(* CODESYS project p6lib-common.library
   Company: MacGregor
   DefaultNamespace: p6com
   Version: 1.1.4
   DocFormat: reStructuredText
   Placeholder: p6lib_common
   Title: p6lib_common

Project tree, tasks and I/O mapping:
  libraries: p7lib-basetypes, * (MacGregor); Tc2_EtherCAT, * (Beckhoff Automation GmbH); Tc2_Math, * (Beckhoff Automation GmbH); Tc2_Standard, * (Beckhoff Automation GmbH); Tc2_System, * (Beckhoff Automation GmbH); Tc2_Utilities, * (Beckhoff Automation GmbH); Tc3_EventLogger, * (Beckhoff Automation GmbH); Tc3_Module, * (Beckhoff Automation GmbH)
  AnalogOut/
    DUT/
      data type EL40xxIO_out
    function block AnalogOutBiPolarScalableAA [ST]: processing
    function block AnalogOutEL40xx [ST]: processing, Value
    function block AnalogOutPercentAA [ST]: processing
    function block AnalogOutUniPolarScalableAA [ST]: processing
    OutputClassCatalog.txt
  00000000-0000-0000-0000-000000000000|AnalogOut\OutputClassCatalog.txt
  ByteAndBits/
    function ClearBit16 [ST]
    function ClearBit8 [ST]
    function Get_LSB_From_UINT [ST]
    function Get_LSB_From_Word [ST]
    function Get_MSB_From_UINT [ST]
    function Get_MSB_From_Word [ST]
    function GetBit16 [ST]
    function GetBit8 [ST]
    function SetBit16 [ST]
    function SetBit8 [ST]
  Concurrency/
    interface IMutex: acquire, acquired, context, isAcquiredByMe, release
    function block Mutex [ST]: acquire, acquired, context, isAcquiredByMe, release
  counter/
    function block CounterExpansion [ST]: FromDINT_TO_LINT
  Cycle Time/
    function block CycleTime [ST]: Cycletime, update
  EmergencyStop/
    DUT/
      data type ConfigEmergencyStop
      data type EStopSM
    function block EmergencyStop [ST]: Activated, ActivatedSwitchIdx, ActivatedSwitchName, ExternEStop, GroupError, resetGroupError
  EventManagement/
    DUT/
      data type AlarmTable
      data type EventProcessing
    function block AlarmAnalog [ST]: _createArguments, _processing, _processPipeline
    function block AlarmAnalogValueHigh [ST]: _processPipeline
    function block AlarmAnalogValueLow [ST]: _processPipeline
    function block AlarmCollector [ST]: AlarmCritical, AlarmWarning, ConfirmAlarms, OnAlarmConfirmed, OnAlarmRaised, reset, update
    function block AlarmCollectorEx [ST]: AlarmCritical, AlarmWarning, ConfirmAlarms, copyTableToHMI, delEvent, Execute, getText, insertEvent, OnAlarmCleared, OnAlarmConfirmed, OnAlarmRaised, reset
    function block AlarmDigital [ST]
    function block AlarmDigitalEx [ST]: _createArguments
    function block AlarmEvent [ST]: _createArguments, _createEvent, clear, confirm, FB_init, raise, Raised
    function block AlarmOilFilter [ST]
    function block AlarmSensorError [ST]
    function block AlarmSensorValueHigh [ST]: _processPipeline
    function block AlarmSensorValueLow [ST]: _processPipeline
    function block AlarmSimple [ST]
    function block StartupDelay [ST]: Done, FB_init
  Fieldbus/
    DUT/
      data type CU2508StatIO_In
      data type EFieldbusQueryResult
      data type ESimpleFieldbusSM
      data type EthercatCoEObject
      data type EthercatCoEObjectArray
      data type EthercatCoEValueArray
      data type EthTypes
      data type EthValue
      data type EthWriteCoEArraySM
    function block Ethercat [ST]: _readCoEData, _writeCoEData, isDevice, readCoEDataBYTE, readCoEDataDINT, readCoEDataDWORD, readCoEDataINT, readCoEDataLINT, readCoEDataLREAL, readCoEDataLWORD, readCoEDataREAL, readCoEDataSINT, readCoEDataUDINT, readCoEDataUINT, readCoEDataULINT, readCoEDataUSINT, readCoEDataWORD, readCoEValueArray, wait, writeCoEDataBYTE, writeCoEDataDINT, writeCoEDataDWORD, writeCoEDataINT, writeCoEDataLINT, writeCoEDataLREAL, writeCoEDataLWORD, writeCoEDataREAL, writeCoEDataSINT, writeCoEDataUDINT, writeCoEDataUINT, writeCoEDataULINT, writeCoEDataUSINT, writeCoEDataWORD, writeCoEValueArray
    function block EthercatCU2508Stat [ST]: getLostFrames, setNull
    function block EthercatMasterStat [ST]: LostFrames, setNull
  IOHandler/
    interface IIOHandler: get
    function block IOHandler [ST]: FB_init, get
  Math/
    function CosineRuleKnownAllSides [ST]
    function CosineRuleKnownAnAngle [ST]
    function HorizontalLength [ST]
    function Scale [ST]
    function Signum [ST]
    function VerticalHeight [ST]
  MRU/
    DUT/
      data type ConfigMRU
    interface IMRUReader: DataAvailable, getData
    function block MRU [ST]: getValues, transform, update
  NMEA/
    DUT/
      data type TNMEAint
      data type TNMEAreal
      data type TNMEAsentence
      data type TNMEAstring
      data type TNMEAStructDescription
    function block NMEA_TrawlLength [ST]
    function block NMEA_TrawlSpeed [ST]
    function block NMEA_TrawlTension [ST]
    function block NMEAParser [ST]: _hexChkSum_to_byte, _incp, calcChkSum, getChkSumFromSentence, getHeader, getIntField, getRealField, getStringField, parse, setFieldsOfInterest
    function block NMEASentence [ST]: calcCheckSum, DataOut, formatSentenceWith3Values
    function block NMEATransmitter6021 [ST]: Busy
  ObjectProtocols/
    DUT/
    V1/
      function block ProtoBase1ToN [ST]: attach, FB_init, getNoServices, getService, getServiceByIdx, isAttached, resetService, setService
      function block ProtoBaseNTo1 [ST]: attach, FB_init, getMaster, getMasterByIdx, getNoMasters, isAttached, resetServices, setMaster
      function block ProtoMasterSingleService [ST]: attach, getService
  OperationTime/
    DUT/
      data type OperationTimeSM
    function block DeviceOpTime [ST]: Optime
    function block OperationTimeCounter [ST]: reset, update
  ParameterManagment/
    AddParameter/
      function block AddParameterBool [ST]
      function block AddParameterInt [ST]
      function block AddParameterLreal [ST]
      function block AddParameterStr [ST]
      function block AddParameterTime [ST]
    DUT/
      data type DataType
      data type ParameterList
  PID/
    DUT/
    function block HTrawlController [ST]: ErrorPosition, ErrorVelocity, Tension, TorqueOut
    function block HTrawlController2 [ST]: CtrlLimit, ErrorPosition, ErrorVelocity, Tension, TorqueOut, VelocitySetpoint
    function block HTrawlController3 [ST]: CtrlLimit, ErrorPosition, ErrorVelocity, Tension, TorqueOut, VelocitySetpoint
    function block HTrawlController4 [ST]: CtrlLimit, ErrorPosition, ErrorVelocity, Tension, TorqueOut, VelocitySetpoint
    function block HTrawlController5 [ST]: CtrlLimit, ErrorPosition, ErrorVelocity, Tension, TorqueOut, VelocitySetpoint
    function block HTrawlController6 [ST]: CtrlLimit, ErrorPosition, ErrorVelocity, Tension, TorqueOut, VelocitySetpoint
    function block PIDController [ST]: Error, Out, update
    function block PIDController2P [ST]: Error, Out, update
    function block PIDControllerLINT [ST]: Error, Out, update
  Sensor/
    DUT/
      data type BarthUnsignedIO_In
      data type EL30xxIO_in
      data type EL30xxStatus
      data type EL30xxStatusWordBit
      data type SensorBinaryIO_in
    Fishpump/
      DUT/
        data type SensorBarthIO_In
      function block SensorBarthBase [ST]: Error, processing, Value, ValueRaw
      function block SensorBarthPressure [ST]: processing
      function block SensorBarthTemp [ST]: processing
      function block SensorBarthUnsigned [ST]: processing
    HandlingBody/
      function block AnglePosition [ST]: processing
      function block StrokePosition [ST]: Angle, Height, Length, processing, Stroke
      data type StrokePositionConfig
    HydPressure/
      data type AnglePositionConfig
      function block HydPressure250barAA [ST]: processing
      function block HydPressure60barAA [ST]: processing
    OilFilter/
      function block OilFilterSensor [ST]: Error, processing, Value, ValueRaw
    Pressure/
      function block Pressure10barAA [ST]: processing
    Scalable/
      function block Sensor20mAA [ST]: processing
      function block SensorASymRangeAA [ST]: processing
      function block SensorSymRange [ST]: processing
      function block SensorSymRangeAA [ST]: processing
    Temperature/
      function block TempSensorAB [ST]: processing
      function block TempSensorAC [ST]: processing
      function block TempSensorAA [ST]: processing
    function block DummySensor [ST]: Error, Value, ValueRaw
    SensorCatalog.txt
    function block SensorEL30xx [ST]: Error, processing, Value, ValueRaw
  00000000-0000-0000-0000-000000000000|Sensor\SensorCatalog.txt
  SignalClassifier/
    DUT/
    function block SignalClassGTEQ [ST]: processing, Signal, update
    function block SignalClassLTEQ [ST]: processing, Signal, update
  SignalProcessing/
    DUT/
      data type SwitchHysteresisSM
    function block Filter1stDeg [ST]
    function block Filter1stDegEx [ST]: reset
    function block InverseOneSideTest [ST]
    interface ISignalPipeline: analogAbs, analogFilter1stDeg, analogLimitBand, analogLimitLowerBoundary, analogLimitUpperBoundary, analogReversePolarity, analogScale, boolInverse, boolTestTimeSpan, getAnalogValue, getBinaryValue, retrieveValues, setBoolInput, setLRealInput, testFalling, testGreaterOrEqual, testLessOrEqual, testRaising
    function block OneSideTest [ST]
    function block SignalPipeline [ST]: analogAbs, analogFilter1stDeg, analogLimitBand, analogLimitLowerBoundary, analogLimitUpperBoundary, analogReversePolarity, analogScale, boolInverse, boolTestTimeSpan, getAnalogValue, getBinaryValue, retrieveValues, setBoolInput, setLRealInput, testFalling, testGreaterOrEqual, testLessOrEqual, testRaising
    function block TwoSideTest [ST]
  Signals/
    function block OneShotSignal [ST]: Get, Set
    function block OneShotSignalInt [ST]: Get, Set
  TimingGenerators/
    function block CycleGenerator [ST]: Q, update
    function block CycleTimer [ST]
    function block SymmetricPulse [ST]: Value
  UnitConversion/
    DUT/
      data type ConfigSystemUnits
      data type LengthUnits
      data type TensionUnits
      data type VelocityUnits
    function block UnitConverter [ST]: getLengthUnit, getTensionUnit, getVelocityUnit, kgToUnit, meterToUnit, MSToUnit, unitToKg, unitToMeter, unitToMS
  global variables Parameters
*)

// AnalogOut/DUT/EL40xxIO_out
TYPE EL40xxIO_out :
	STRUCT
		output	: INT;
	END_STRUCT
END_TYPE

// EmergencyStop/DUT/ConfigEmergencyStop
TYPE ConfigEmergencyStop :
	STRUCT
		switchname : ARRAY[0..Parameters.SizeOfEStopArray-1] OF P6IdName;
	END_STRUCT
END_TYPE

// EmergencyStop/DUT/EStopSM
{attribute 'qualified_only'}
{attribute 'strict'}
TYPE EStopSM :
	(
		STARTUP 			:= 0,
		WAITRESET			:= 10,
		IDLE				:= 20,
		ESTOP				:= 30,
		ESTOP_RELEASED		:= 40,
		GRP_RST_START		:= 50,
		GRP_RST_EXE			:= 60, 
		GRP_RST_END			:= 70
	) INT;
END_TYPE

// EventManagement/DUT/AlarmTable
TYPE AlarmTable :
	STRUCT
		eventID : UDINT;
		timestamp : STRING;
		message : STRING(255);
	END_STRUCT
END_TYPE

// EventManagement/DUT/EventProcessing
TYPE EventProcessing :
	STRUCT
		event : REFERENCE TO FB_TcEvent;
		uid : UDINT;
		eventID : UDINT;
		timestamp : STRING;
		message : STRING(255);
		hasTxt : BOOL;
	END_STRUCT
END_TYPE

// Fieldbus/DUT/CU2508StatIO_In
TYPE CU2508StatIO_In :
	STRUCT
		addr : ARRAY[0..7] OF AMSNETID;
	END_STRUCT
END_TYPE

// Fieldbus/DUT/EFieldbusQueryResult
{attribute 'qualified_only'}
{attribute 'strict'}
TYPE EFieldbusQueryResult :
(
	OK 					:= 0,
	FAIL				:= -1,
	BUSY				:= 1
) INT;
END_TYPE

// Fieldbus/DUT/ESimpleFieldbusSM
{attribute 'qualified_only'}
{attribute 'strict'}
TYPE ESimpleFieldbusSM :
(
	IDLE			:= 0,
	STARTUP			:= 1,
	WAITONRESULT	:= 2,
	RESULT			:= 3			
) INT;
END_TYPE

// Fieldbus/DUT/EthercatCoEObject
TYPE EthercatCoEObject :
	STRUCT
		para	: DWORD := 16#FFFF_FFFF; // Format XXXXYY X: Parameter group, Y: Parameter. Has no functionality other than to provide data for the HMI and to mark the end of the list
		idx		: WORD;
		sidx	: BYTE;  
		tclass 	: EthTypes := EthTypes.TWORD;	
	END_STRUCT
END_TYPE

// Fieldbus/DUT/EthercatCoEObjectArray
TYPE 
	EthercatCoEObjectArray : ARRAY[0..Parameters.SizeOfEthCoEValues-1] OF EthercatCoEObject; 
END_TYPE

// Fieldbus/DUT/EthercatCoEValueArray
TYPE 
	EthercatCoEValueArray : ARRAY[0..Parameters.SizeOfEthCoEValues-1] OF EthValue; 
END_TYPE

// Fieldbus/DUT/EthTypes
{attribute 'qualified_only'}
{attribute 'strict'}
TYPE EthTypes :
(
	TWORD			:= 0,
	TBYTE			:= 1,
	TDWORD			:= 2,
	TLWORD			:= 3,
	TSINT			:= 4,
	TUSINT			:= 5,
	TINT			:= 6,
	TUINT			:= 7,
	TDINT			:= 8,
	TUDINT			:= 9,
	TLINT			:= 10,
	TULINT			:= 11,
	TREAL			:= 12,
	TLREAL			:= 13
) INT;
END_TYPE

// Fieldbus/DUT/EthValue
TYPE EthValue :
	UNION
		VBYTE			: BYTE;
		VWORD			: WORD;
		VDWORD			: DWORD;
		VLWORD			: LWORD;
		VSINT			: SINT;
		VUSINT			: USINT;
		VINT			: INT;
		VUINT			: UINT;
		VDINT			: DINT;
		VUDINT			: UDINT;
		VLINT			: LINT;
		VULINT			: ULINT;
		VREAL			: REAL;
		VLREAL			: LREAL;
	END_UNION
END_TYPE

// Fieldbus/DUT/EthWriteCoEArraySM
{attribute 'qualified_only'}
{attribute 'strict'}
TYPE EthWriteCoEArraySM :
(
	IDLE		 	:= 0,
	WRITE			:= 10,
	ERROR			:= 20,
	READY			:= 30,
	INCR			:= 40
) INT;
END_TYPE

// MRU/DUT/ConfigMRU
TYPE ConfigMRU :
	STRUCT
		Option_Transformation		: BOOL := FALSE;
		Option_Reverse_Position 	: BOOL := FALSE;
		Option_Reverse_Velocity 	: BOOL := FALSE;
		Option_Reverse_Acceleration : BOOL := FALSE;
		Option_Reverse_Roll			: BOOL := FALSE;
		Option_Reverse_Ritch		: BOOL := FALSE;
		Option_MRUSet				: INT  := -1; // Values for coordinate set from 0..9, when transformation is used
				
		// Section Transformation 					
		CycleTime 					: LREAL := 0.05; // Cycletime of the MRU in sec
		FilterAcceleration			: LREAL := 1.0; // Values from 0..1!
		PosX						: ARRAY[0..19] OF LREAL; // X axis forward aligned
		PosY 						: ARRAY[0..19] OF LREAL; // Y axis port aliged
		PosZ						: ARRAY[0..19] OF LREAL; // Z upwards aligned
	END_STRUCT
END_TYPE

// NMEA/DUT/TNMEAint
TYPE TNMEAint : LINT; END_TYPE

// NMEA/DUT/TNMEAreal
TYPE TNMEAreal : LREAL; END_TYPE

// NMEA/DUT/TNMEAsentence
TYPE TNMEAsentence : STRING(254); END_TYPE

// NMEA/DUT/TNMEAstring
TYPE TNMEAstring : STRING(128); END_TYPE

// NMEA/DUT/TNMEAStructDescription
TYPE TNMEAStructDescription : STRING(32); END_TYPE

// OperationTime/DUT/OperationTimeSM
{attribute 'qualified_only'}
{attribute 'strict'}
TYPE OperationTimeSM :
(
	IDLE 		:= 0,
	ACTIVE		:= 1
);
END_TYPE

// ParameterManagment/DUT/DataType
TYPE DataType :
	STRUCT
		intType : INT;
		boolType : BOOL;
		stringType : STRING;
		lrealType : LREAL;
		timeType : TIME;
	END_STRUCT
END_TYPE

// ParameterManagment/DUT/ParameterList
TYPE ParameterList :
	STRUCT
		name : STRING := 'Ω FREE';
		value : DataType;
		unit : STRING;
		status : STRING;
	END_STRUCT
END_TYPE

// Sensor/DUT/BarthUnsignedIO_In
TYPE BarthUnsignedIO_In :
	STRUCT
		input	: INT;
	END_STRUCT
END_TYPE

// Sensor/DUT/EL30xxIO_in
TYPE EL30xxIO_in :
	STRUCT
		status 	: EL30xxStatus;
		input	: INT;
	END_STRUCT
END_TYPE

// Sensor/DUT/EL30xxStatus
TYPE EL30xxStatus :
	UNION
		twobyte : WORD;
		bits 	: EL30xxStatusWordBit;
	END_UNION
END_TYPE

// Sensor/DUT/EL30xxStatusWordBit
TYPE EL30xxStatusWordBit :
	STRUCT
		UnderRange			: BIT;		// 0
		OverRange			: BIT;		// 1
		Limit1				: BIT;		// 2
		Limit2				: BIT;		// 3
		Reserved4			: BIT;		// 4
		Reserved5			: BIT;		// 5
		Error				: BIT;		// 6
		Reserved7			: BIT;		// 7
		Reserved8			: BIT;		// 8
		Reserved9			: BIT;		// 9	
		Reserved10			: BIT;		// 10
		Reserved11			: BIT;		// 11
		Reserved12			: BIT;		// 12
		Reserved13			: BIT;		// 13
		Reserved14			: BIT;		// 14
		Reserved15			: BIT;		// 15
	END_STRUCT
END_TYPE

// Sensor/DUT/SensorBinaryIO_in
TYPE SensorBinaryIO_in :
	STRUCT
		signal	: BOOL; 
	END_STRUCT
END_TYPE

// Sensor/Fishpump/DUT/SensorBarthIO_In
TYPE SensorBarthIO_In :
	STRUCT
		input	: WORD;
	END_STRUCT
END_TYPE

// Sensor/HandlingBody/StrokePositionConfig
TYPE StrokePositionConfig :
	STRUCT
		FilterCoefficient : LREAL := 0.1;// 1stDegFilter, cant be 0.
		CalibratedLowerLimit : LREAL;	//min sensor measurement
		CalibratedUpperLimit : LREAL;	//max sensor measurement
		MinStroke : LREAL;
		MaxStroke : LREAL;
		CylinderToNextJointMin : LREAL;
		CylinderToNextJointMax : LREAL;	
		
		BoltToBoltLength : LREAL;
		BoltToCylinderBoltLength : LREAL;
		TiltLegLength : LREAL;
		InverseDirection : BOOL;
	END_STRUCT
END_TYPE

// Sensor/HydPressure/AnglePositionConfig
TYPE AnglePositionConfig :
	STRUCT
		FilterCoefficient : LREAL := 0.1;// 1stDegFilter, cant be 0.
		CalibratedLowerLimit : LREAL;	//min sensor measurement
		CalibratedUpperLimit : LREAL;	//max sensor measurement
		MaxAngle : LREAL;		// [deg]total range this joint operate in
	END_STRUCT
END_TYPE

// SignalProcessing/DUT/SwitchHysteresisSM
{attribute 'qualified_only'}
{attribute 'strict'}
TYPE SwitchHysteresisSM :
(
	START 			:= 0,
	IDLE			:= 10,
	ON				:= 20,
	WAITFOROFF		:= 30,
	BANDUP			:= 40,
	BANDDOWN		:= 50 
) INT;
END_TYPE

// UnitConversion/DUT/ConfigSystemUnits
TYPE ConfigSystemUnits :
	STRUCT
		velocityUnit : VelocityUnits;
		tensionUnit  : TensionUnits;
		lengthUnit   : LengthUnits;
	END_STRUCT
END_TYPE

// UnitConversion/DUT/LengthUnits
{attribute 'qualified_only'}
{attribute 'strict'}
TYPE LengthUnits :
(
	METER 	:= 0,
	FEET 	:= 1,
	FATHOM 	:= 2
) DINT;
END_TYPE

// UnitConversion/DUT/TensionUnits
{attribute 'qualified_only'}
{attribute 'strict'}
TYPE TensionUnits :
(
	KILO 		:= 0,
	TON_METRIC	:= 1,
	TON_IMPERIAL:= 2,
	POUND 		:= 3
) DINT;
END_TYPE

// UnitConversion/DUT/VelocityUnits
{attribute 'qualified_only'}
{attribute 'strict'}
TYPE VelocityUnits :
(
	METER_PER_SEC 	:= 0,
	METER_PER_MIN 	:= 1,
	FEET_PER_MIN 	:= 2,
	FATHOM_PER_MIN	:= 3
) DINT;
END_TYPE

// Parameters
{attribute 'qualified_only'}
VAR_GLOBAL CONSTANT
	SizeOfEthCoEValues 	: INT := 200;
	SizeOfEStopArray	: INT := 100;
	
	//
	// This is related to protocol definitions
	//
	ServicesPerMaster	: DINT := 100;
	MastersPerService	: DINT := 100;
END_VAR

// AnalogOut/AnalogOutBiPolarScalableAA
(* 
	Use this class only, when the scaling values are unknown!
*)
FUNCTION_BLOCK AnalogOutBiPolarScalableAA EXTENDS AnalogOutEL40xx IMPLEMENTS IAnalogOut
VAR_INPUT
	ValueMax	: LREAL;
	ValueMin	: LREAL;
END_VAR
VAR
	{attribute 'hide'} 
	pipe			: SignalPipeline;
END_VAR

SUPER^();
THIS^.processing();

METHOD PROTECTED  processing : BOOL
VAR_INST
	val : LREAL;
END_VAR
IF ABS(ValueMax-ValueMin)>=0.1 THEN
	val :=  THIS^.pipe
						.setLRealInput(THIS^.rvalue)
						.analogScale(ValueMin, ValueMax, THIS^.ADC_VALUE_MIN, THIS^.ADC_VALUE_MAX, TRUE)
						.getAnalogValue();
								
	THIS^.IO_Out.output := LREAL_TO_INT(val);
ELSE
	THIS^.IO_Out.output := 0;	
END_IF
END_METHOD

END_FUNCTION_BLOCK

// AnalogOut/AnalogOutEL40xx
FUNCTION_BLOCK ABSTRACT AnalogOutEL40xx
VAR_INPUT
	IO_Out					: REFERENCE TO EL40xxIO_Out;
END_VAR
VAR
	{attribute 'hide'} 
	rvalue					: LREAL;							
END_VAR
VAR CONSTANT
	{attribute 'hide'} 
	ADC_VALUE_MAX 			: LREAL := 16#7FFF;
	{attribute 'hide'} 
	ADC_VALUE_MIN 			: LREAL := 0;
END_VAR

METHOD PROTECTED ABSTRACT processing : BOOL
END_METHOD

{attribute 'monitoring' := 'call'}
{attribute 'TcRpcEnable'}
PROPERTY Value : LREAL
SET
rvalue := Value;
END_SET
END_PROPERTY

END_FUNCTION_BLOCK

// SignalProcessing/SignalPipeline
{attribute 'hide_all_locals'}
FUNCTION_BLOCK SignalPipeline IMPLEMENTS ISignalPipeline
VAR
	// Internal processing
	process_value_lreal				: LREAL;
	process_value_bool				: BOOL;
END_VAR

METHOD analogAbs : ISignalPipeline
VAR_INPUT
	Value 		: LREAL;
END_VAR
THIS^.process_value_lreal := ABS(THIS^.process_value_lreal);

analogAbs := THIS^;
END_METHOD

METHOD analogFilter1stDeg : ISignalPipeline
VAR_INPUT
	Coefficient				: LREAL;
END_VAR
VAR_INST
	_filter1stDeg 					: Filter1stDeg;	
END_VAR
_filter1stDeg( 
			Value:= THIS^.process_value_lreal, 
			Coefficient:= Coefficient, 
			Out => THIS^.process_value_lreal
		);

analogFilter1stDeg := THIS^;
END_METHOD

METHOD analogLimitBand : ISignalPipeline
VAR_INPUT
	BoundaryLower 		: LREAL;
	BoundaryUpper 		: LREAL;
END_VAR
THIS^.process_value_lreal := LIMIT(BoundaryLower, THIS^.process_value_lreal, BoundaryUpper);

analogLimitBand := THIS^;
END_METHOD

METHOD analogLimitLowerBoundary : ISignalPipeline
VAR_INPUT
	Boundary 		: LREAL;
END_VAR
THIS^.process_value_lreal := MAX(Boundary, THIS^.process_value_lreal);

analogLimitLowerBoundary := THIS^;
END_METHOD

METHOD analogLimitUpperBoundary : ISignalPipeline
VAR_INPUT
	Boundary 		: LREAL;
END_VAR
THIS^.process_value_lreal := MIN(Boundary, THIS^.process_value_lreal);

analogLimitUpperBoundary := THIS^;
END_METHOD

METHOD analogReversePolarity : ISignalPipeline
VAR_INPUT
	Enable : BOOL;
END_VAR
THIS^.process_value_lreal := SEL(Enable, THIS^.process_value_lreal, -THIS^.process_value_lreal);

analogReversePolarity := THIS^;
END_METHOD

METHOD analogScale : ISignalPipeline
VAR_INPUT
	InputMin 		: LREAL;
	InputMax		: LREAL;
	OutputMin		: LREAL;
	OutputMax		: LREAL;
	LimitOutput		: BOOL;
END_VAR
THIS^.process_value_lreal := Scale(
									Value 		:= THIS^.process_value_lreal,
									InputMin 	:= InputMin,
									InputMax	:= InputMax,
									OutputMin	:= OutputMin,
									OutputMax	:= OutputMax,
									LimitOutput	:= LimitOutput 
								);
								
analogScale := THIS^;
END_METHOD

METHOD boolInverse : ISignalPipeline

THIS^.process_value_bool := NOT THIS^.process_value_bool;

boolInverse := THIS^;
END_METHOD

METHOD boolTestTimeSpan : ISignalPipeline
VAR_INPUT
	TimeSpan	: TIME;
END_VAR
VAR_INST
	timerOn 	: TON;
END_VAR

timerOn(IN := THIS^.process_value_bool, PT := TimeSpan);

THIS^.process_value_bool := timerOn.Q;

boolTestTimeSpan := THIS^;
END_METHOD

METHOD getAnalogValue : LREAL

getAnalogValue := THIS^.process_value_lreal;
END_METHOD

METHOD getBinaryValue : BOOL

getBinaryValue := THIS^.process_value_bool;
END_METHOD

METHOD retrieveValues : ISignalPipeline
VAR_INPUT
	ValueLReal 	: REFERENCE TO LREAL;
	ValueBool	: REFERENCE TO BOOL;
END_VAR
IF  __ISVALIDREF(ValueLReal) THEN
	ValueLReal := THIS^.process_value_lreal;
END_IF

IF  __ISVALIDREF(ValueBool) THEN
	ValueBool := THIS^.process_value_bool;
END_IF

retrieveValues := THIS^;
END_METHOD

METHOD setBoolInput : ISignalPipeline
VAR_INPUT
	Value : BOOL;
END_VAR
THIS^.process_value_bool := Value;

setBoolInput := THIS^;
END_METHOD

(*
This method has to get the raw value and put into internal_processing_value 
when THIS^.retrieve = TRUE 
*)
METHOD setLRealInput : ISignalPipeline
VAR_INPUT
	Value	: LREAL;
END_VAR
THIS^.process_value_lreal := Value;
THIS^.process_value_bool := FALSE;


setLRealInput := THIS^;
END_METHOD

METHOD testFalling : ISignalPipeline
VAR_INST
	trigger : F_TRIG;
END_VAR
trigger(CLK := THIS^.process_value_bool, Q=>THIS^.process_value_bool);

testFalling := THIS^;
END_METHOD

METHOD testGreaterOrEqual : ISignalPipeline
VAR_INPUT
	Value		: LREAL;
	Hysteresis	: LREAL;
	MakeAnd		: BOOL;
END_VAR
VAR_INST
	oneside		: OneSideTest;
	res 		: BOOL;
END_VAR
oneside(
			Level := Value,
			Hysteresis := Hysteresis, 
			Value		:= THIS^.process_value_lreal,
			Out => res
		);
					
THIS^.process_value_bool := SEL(
								MakeAnd, 
								res OR THIS^.process_value_bool, 
								res AND THIS^.process_value_bool
							);
							
testGreaterOrEqual := THIS^;
END_METHOD

METHOD testLessOrEqual : ISignalPipeline
VAR_INPUT
	Value		: LREAL;
	Hysteresis	: LREAL;
	MakeAnd		: BOOL;
END_VAR
VAR_INST
	inv_oneside		: InverseOneSideTest;
	res 			: BOOL;
END_VAR
inv_oneside(
				Level 		:= Value,
				Hysteresis 	:= Hysteresis, 
				Value		:= THIS^.process_value_lreal,
				Out 		=> res
			);
					
THIS^.process_value_bool := SEL(
								MakeAnd, 
								res OR THIS^.process_value_bool, 
								res AND THIS^.process_value_bool
							);
							
							
testLessOrEqual := THIS^;
END_METHOD

METHOD testRaising : ISignalPipeline
VAR_INST
	trigger : R_TRIG;
END_VAR
trigger(CLK := THIS^.process_value_bool, Q=>THIS^.process_value_bool);

testRaising := THIS^;
END_METHOD

END_FUNCTION_BLOCK

// SignalProcessing/ISignalPipeline
INTERFACE ISignalPipeline

METHOD analogAbs : ISignalPipeline
VAR_INPUT
	Value 		: LREAL;
END_VAR
END_METHOD

METHOD analogFilter1stDeg : ISignalPipeline
VAR_INPUT
	Coefficient				: LREAL;
END_VAR
END_METHOD

METHOD analogLimitBand : ISignalPipeline
VAR_INPUT
	BoundaryLower 		: LREAL;
	BoundaryUpper 		: LREAL;
END_VAR
END_METHOD

METHOD analogLimitLowerBoundary : ISignalPipeline
VAR_INPUT
	Boundary 		: LREAL;
END_VAR
END_METHOD

METHOD analogLimitUpperBoundary : ISignalPipeline
VAR_INPUT
	Boundary 		: LREAL;
END_VAR
END_METHOD

METHOD analogReversePolarity : ISignalPipeline
VAR_INPUT
	Enable : BOOL;
END_VAR
END_METHOD

METHOD analogScale : ISignalPipeline
VAR_INPUT
	InputMin 		: LREAL;
	InputMax		: LREAL;
	OutputMin		: LREAL;
	OutputMax		: LREAL;
	LimitOutput		: BOOL;
END_VAR
END_METHOD

METHOD boolInverse : ISignalPipeline
END_METHOD

METHOD boolTestTimeSpan : ISignalPipeline
VAR_INPUT
	TimeSpan	: TIME;
END_VAR
END_METHOD

METHOD getAnalogValue : LREAL
END_METHOD

METHOD getBinaryValue : BOOL
END_METHOD

METHOD retrieveValues : ISignalPipeline
VAR_INPUT
	ValueLReal 	: REFERENCE TO LREAL;
	ValueBool	: REFERENCE TO BOOL;
END_VAR
END_METHOD

METHOD setBoolInput : ISignalPipeline
VAR_INPUT
	Value : BOOL;
END_VAR
END_METHOD

(*
This method has to get the raw value and put into internal_processing_value 
when THIS^.retrieve = TRUE 
*)
METHOD setLRealInput : ISignalPipeline
VAR_INPUT
	Value : LREAL;
END_VAR
END_METHOD

METHOD testFalling : ISignalPipeline
END_METHOD

METHOD testGreaterOrEqual : ISignalPipeline
VAR_INPUT
	Value		: LREAL;
	Hysteresis	: LREAL;
	MakeAnd		: BOOL;
END_VAR
END_METHOD

METHOD testLessOrEqual : ISignalPipeline
VAR_INPUT
	Value		: LREAL;
	Hysteresis	: LREAL;
	MakeAnd		: BOOL;
END_VAR
END_METHOD

METHOD testRaising : ISignalPipeline
END_METHOD

END_INTERFACE

// SignalProcessing/Filter1stDeg
(*
Purpose
=======
This is a 1st deg filter class. The coeffcient has a range from 0..1 and is limited automagically by this class

Methods And Properties
======================
*)
{attribute 'hide_all_locals'}
FUNCTION_BLOCK Filter1stDeg
VAR_INPUT
	Value 			: LREAL;
	Coefficient  	: LREAL;
END_VAR
VAR_OUTPUT
	Out 			: LREAL; 
END_VAR
VAR
	value_1 		: LREAL;
	value_0			: LREAL;
	CoefficientCopy : LREAL;
END_VAR


CoefficientCopy := LIMIT(0.0, Coefficient, 1.0);
value_0 := Value * CoefficientCopy + (1.0 - CoefficientCopy) * value_1; 

value_1 := value_0;

Out 	:= value_0;

END_FUNCTION_BLOCK

// Math/Scale
(*
This function is transposing an input range to an output range. The option of 
limiting output is for cases when a full range calibration isn't possible 
*)
{attribute 'hide_all_locals'}
FUNCTION Scale : LREAL
VAR_INPUT
	Value			: LREAL;
	InputMin 		: LREAL;
	InputMax 		: LREAL;
	OutputMin 		: LREAL;
	OutputMax 		: LREAL;
	LimitOutput : BOOL;
END_VAR
VAR
END_VAR

IF ((InputMax - InputMin) <> 0) THEN
	Scale := (OutputMax - OutputMin) / (InputMax - InputMin) * (Value - InputMin) + OutputMin;
	IF LimitOutput THEN
		IF OutputMax >= OutputMin THEN 
			Scale := LIMIT(OutputMin, Scale, OutputMax);
		ELSE
			Scale := LIMIT(OutputMax, Scale, OutputMin);			
		END_IF
	END_IF
ELSE
	Scale := 0;
END_IF

END_FUNCTION

// SignalProcessing/OneSideTest
(*
Purpose
=======
This class is a test whether a value is outside a range from 0 ..max. The max value has
a hysteresis



Methods And Properties
======================
*)
{attribute 'hide_all_locals'}
FUNCTION_BLOCK OneSideTest
VAR_INPUT
	Level	 	: LREAL;
	Hysteresis	: LREAL;
	Value		: LREAL;
END_VAR
VAR_OUTPUT
	Out			: BOOL;
END_VAR
VAR
	state : SwitchHysteresisSM;
END_VAR


CASE state OF 
	SwitchHysteresisSM.START:
		state := SwitchHysteresisSM.IDLE; 
		
	SwitchHysteresisSM.IDLE:
		IF Value >= Level + ABS(Hysteresis/2.0) THEN
			state := SwitchHysteresisSM.ON;
		END_IF
	
	SwitchHysteresisSM.ON:
		IF Value <= Level - ABS(Hysteresis/2.0) THEN
			state := SwitchHysteresisSM.IDLE;
		END_IF
	ELSE
		state := SwitchHysteresisSM.START;
END_CASE


Out := state = SwitchHysteresisSM.ON;

END_FUNCTION_BLOCK

// SignalProcessing/InverseOneSideTest
(*
Purpose
=======
This class is a test whether a value is outside a range from 0 ..max. The max value has
a hysteresis

Methods And Properties
======================
*)
{attribute 'hide_all_locals'}
FUNCTION_BLOCK InverseOneSideTest
VAR_INPUT
	Level	 	: LREAL;
	Hysteresis	: LREAL;
	Value		: LREAL;
END_VAR
VAR_OUTPUT
	Out 		: BOOL;
END_VAR
VAR
	state : SwitchHysteresisSM;
END_VAR


CASE state OF 
	SwitchHysteresisSM.START:
		state := SwitchHysteresisSM.IDLE; 
		
	SwitchHysteresisSM.IDLE:
		IF Value <= Level - ABS(Hysteresis/2.0) THEN
			state := SwitchHysteresisSM.ON;
		END_IF
	
	SwitchHysteresisSM.ON:
		IF Value >= Level + ABS(Hysteresis/2.0) THEN
			state := SwitchHysteresisSM.IDLE;
		END_IF
	ELSE
		state := SwitchHysteresisSM.START;
END_CASE


Out :=  state = SwitchHysteresisSM.ON;

END_FUNCTION_BLOCK

// AnalogOut/AnalogOutPercentAA
(* 
	Use this class only, when the scaling values are unknown!
*)
FUNCTION_BLOCK AnalogOutPercentAA EXTENDS AnalogOutEL40xx IMPLEMENTS IAnalogOut
VAR
	{attribute 'hide'} 
	pipe			: SignalPipeline;
END_VAR

SUPER^();
THIS^.processing();

METHOD PROTECTED  processing : BOOL
VAR_INST
	val : LREAL;
END_VAR
val :=  THIS^.pipe
							.setLRealInput(THIS^.rvalue)
							.analogScale(-1.0, 1.0, THIS^.ADC_VALUE_MIN, THIS^.ADC_VALUE_MAX, TRUE)
							.getAnalogValue();
							
THIS^.IO_Out.output := LREAL_TO_INT(val);
END_METHOD

END_FUNCTION_BLOCK

// AnalogOut/AnalogOutUniPolarScalableAA
(* 
	Use this class only, when the scaling values are unknown!
*)
FUNCTION_BLOCK AnalogOutUniPolarScalableAA EXTENDS AnalogOutEL40xx IMPLEMENTS IAnalogOut
VAR_INPUT
	ValueMax	: LREAL;
	ValueMin	: LREAL;
END_VAR
VAR
	{attribute 'hide'} 
	pipe			: SignalPipeline;
END_VAR

SUPER^();
THIS^.processing();

METHOD PROTECTED  processing : BOOL
VAR_INST
	val : LREAL;
END_VAR
IF ABS(ValueMax-ValueMin)>=0.1 THEN
	val :=  THIS^.pipe
								.setLRealInput(THIS^.rvalue)
								.analogScale(ValueMin, ValueMax, 0, THIS^.ADC_VALUE_MAX, TRUE)
								.getAnalogValue();
								
	THIS^.IO_Out.output := LREAL_TO_INT(val);
ELSE
	THIS^.IO_Out.output := 0;	
END_IF
END_METHOD

END_FUNCTION_BLOCK

// ByteAndBits/ClearBit16
FUNCTION ClearBit16 : WORD
VAR_INPUT
	Value 	: WORD;
	N  		: SINT;
END_VAR

ClearBit16 := DWORD_TO_WORD(ClearBit32(Value, N));

END_FUNCTION

// ByteAndBits/ClearBit8
FUNCTION ClearBit8 : BYTE
VAR_INPUT
	Value 	: BYTE;
	N  		: SINT;
END_VAR

ClearBit8 := DWORD_TO_BYTE(ClearBit32(Value, N));

END_FUNCTION

// ByteAndBits/Get_LSB_From_UINT
FUNCTION Get_LSB_From_UINT : USINT
VAR_INPUT
	data : UINT;
END_VAR
VAR
	{attribute 'hide'} 
	p : POINTER TO USINT;
END_VAR

p := ADR(data);
Get_LSB_From_UINT := p^;

END_FUNCTION

// ByteAndBits/Get_LSB_From_Word
FUNCTION Get_LSB_From_Word : BYTE
VAR_INPUT
	data : WORD;
END_VAR
VAR
	{attribute 'hide'} 
	p : POINTER TO BYTE;
END_VAR

p := ADR(data) ;
Get_LSB_From_Word := p^;

END_FUNCTION

// ByteAndBits/Get_MSB_From_UINT
FUNCTION Get_MSB_From_UINT : USINT;
VAR_INPUT
	data : UINT;
END_VAR
VAR
	{attribute 'hide'} 
	p : POINTER TO USINT;
END_VAR

p := ADR(data) + 1;
Get_MSB_From_UINT := p^;

END_FUNCTION

// ByteAndBits/Get_MSB_From_Word
FUNCTION Get_MSB_From_Word : BYTE
VAR_INPUT
	data : WORD;
END_VAR
VAR
	{attribute 'hide'} 
	p : POINTER TO BYTE;
END_VAR

p := ADR(data) + 1;
Get_MSB_From_Word := p^;

END_FUNCTION

// ByteAndBits/GetBit16
FUNCTION GetBit16 : BOOL
VAR_INPUT
	Value 	: WORD;
	N  		: SINT;
END_VAR

GetBit16 := GetBit32(Value, N);

END_FUNCTION

// ByteAndBits/GetBit8
FUNCTION GetBit8 : BOOL
VAR_INPUT
	Value 	: BYTE;
	N  		: SINT;	
END_VAR

GetBit8 := GetBit32(Value, N);

END_FUNCTION

// ByteAndBits/SetBit16
FUNCTION SetBit16 : WORD
VAR_INPUT
	Value 	: WORD;
	N  		: SINT;
END_VAR

SetBit16 := DWORD_TO_WORD(SetBit32(Value, N));

END_FUNCTION

// ByteAndBits/SetBit8
FUNCTION SetBit8 : BYTE;
VAR_INPUT
	Value 	: BYTE;
	N  		: SINT;
END_VAR

SetBit8 := DWORD_TO_BYTE(SetBit32(Value, N));

END_FUNCTION

// Concurrency/IMutex
INTERFACE IMutex

METHOD acquire : BOOL
VAR_INPUT
	Context : DINT;
END_VAR
END_METHOD

PROPERTY acquired : BOOL
GET
END_GET
END_PROPERTY

PROPERTY context : DINT
GET
END_GET
END_PROPERTY

METHOD isAcquiredByMe : BOOL
VAR_INPUT
	Context : DINT;
END_VAR
END_METHOD

METHOD release : BOOL
VAR_INPUT
	Context 	: DINT;
END_VAR
END_METHOD

END_INTERFACE

// Concurrency/Mutex
(*
Purpose
=======
This class is providing a Mutex functionality and is including a context identifier 

Methods And Properties
======================
*)
{attribute 'no_explicit_call' := 'do not call this POU directly'} 
FUNCTION_BLOCK Mutex
VAR
	{attribute 'hide'} 
	_acquired 		: BOOL;
	{attribute 'hide'} 
	_context		: DINT;
END_VAR

METHOD acquire : BOOL
VAR_INPUT
	Context : DINT;
END_VAR
IF NOT _acquired THEN
	acquire 	:= TRUE; 
	_acquired 	:= TRUE;
	_context	:= Context;
ELSE
	acquire 	:= FALSE; 
END_IF
END_METHOD

{attribute 'monitoring' := 'variable'}
PROPERTY acquired : BOOL
GET
acquired := _acquired;
END_GET
END_PROPERTY

{attribute 'monitoring' := 'variable'}
PROPERTY context : DINT
GET
context := _context;
END_GET
END_PROPERTY

METHOD isAcquiredByMe : BOOL
VAR_INPUT
	Context : DINT;
END_VAR

IF _acquired AND (Context = _context) THEN
	isAcquiredByMe := TRUE;
ELSE
	isAcquiredByMe := FALSE;	
END_IF
END_METHOD

METHOD release : BOOL
VAR_INPUT
	Context 	: DINT;
END_VAR
IF _acquired AND (Context=_context) THEN
	_acquired := FALSE;
	release := TRUE;
ELSE
	release := TRUE;	
END_IF
END_METHOD

END_FUNCTION_BLOCK

// counter/CounterExpansion
(*
	This class offers Counter Overflow prevention methods
*) 
FUNCTION_BLOCK CounterExpansion

METHOD FromDINT_TO_LINT : LINT
VAR_INPUT
	Counter 			: DINT;
	Overflow			: REFERENCE TO LINT;
END_VAR
VAR 
	past_counter		: LINT;
	actual_counter		: LINT;
	state 				: DINT;
END_VAR

past_counter := actual_counter;
actual_counter := counter;

CASE state OF 
	0: // no change in range
		IF (past_counter > 0)  AND  (actual_counter < 0) THEN 
			state := 1;
		ELSIF (past_counter < 0) AND (actual_counter > 0) THEN
			state := 2;
		END_IF
		
	1: // overflow on the top
		state := 0;
		Overflow := Overflow + LINT#16#1_0000_0000; 
		
	2: // overflow on the bottom
		state := 0;
		Overflow := Overflow - LINT#16#1_0000_0000; 
END_CASE

FromDINT_TO_LINT := actual_counter + Overflow;
END_METHOD

END_FUNCTION_BLOCK

// Cycle Time/CycleTime
(*
Purpose
=======
This class calculates the cycle time independent of a PLC supplier

Methods And Properties
======================
*)
{attribute 'no_explicit_call' := 'do not call this POU directly'} 
{attribute 'hide_all_locals'}
FUNCTION_BLOCK CycleTime
VAR
	t1, t0 : TIME;
	interval : UDINT;
	_cycletime : LREAL;	
END_VAR

{attribute 'monitoring' := 'variable'}
PROPERTY Cycletime : LREAL
GET
Cycletime := _Cycletime;
END_GET
END_PROPERTY

METHOD update : LREAL
t1 := t0; 

t0 := TIME();

interval := MIN(TIME_TO_UDINT(t0-t1), 100);

_cycletime := MAX(
					UDINT_TO_LREAL(interval)/1000.0,
					0.001
				);


update := _cycletime;
END_METHOD

END_FUNCTION_BLOCK

// EmergencyStop/EmergencyStop
FUNCTION_BLOCK EmergencyStop IMPLEMENTS p7type.IEmergencyStop;
VAR_INPUT
	Enabled									: BOOL;
	Config 									: REFERENCE TO ConfigEmergencyStop; 
END_VAR
VAR
	{attribute 'hide'} started 								: BOOL;
	{attribute 'hide'} state									: EStopSM;
	{attribute 'hide'} startUpTimer							: TON;
						grpResetStart						: TON;
						grpResetExe							: TON;
						grpResetEnd							: TON;
						cycleGen							: SymmetricPulse;
	
	{attribute 'hide'} _resetGroup								: BOOL;	
	{attribute 'hide'} _idx 									: INT;
	
	{attribute 'hide'} _switchIdx 								: INT;  //Switch identifier
	{attribute 'hide'} _switchName								: p7type.P6IdName;

	_EStopSwitches 			AT %I* 			: ARRAY [0..Parameters.SizeOfEStopArray-1] OF BOOL; //Emergency stop input
	_NoEStopDetected 		AT %I* 			: BOOL;	 //Emergency stop signal
	
	_ExternEStop 							: BOOL;
	_TwinSafe_Run 			AT %Q* 			: BOOL := TRUE;  //Run TwinSAFE logic
	_TwinSafeFB_Reset 		AT %Q*			: BOOL;	//Reset emergency stop
	_TwinSafeGroup_Reset	AT %Q*			: BOOL; //Group Reset	
	_TwinSafeGroupErrCom	AT %I*			: BOOL; // Group Com error
	_TwinSafeGroupErrFB		AT %I*			: BOOL; // Group FB Error
	_TwinSafeGroupErrOther	AT %I*			: BOOL; // Group Other Error	
END_VAR

IF NOT started THEN
	started := TRUE;
END_IF

cycleGen(CLK:=T#200MS);
_TwinSafeFB_Reset := cycleGen.Value;

startUpTimer(IN:=(state=EStopSM.WAITRESET), PT:=T#500MS);
grpResetStart(IN:=(state=EStopSM.GRP_RST_START), PT:=T#200MS);
grpResetExe(IN:=(state=EStopSM.GRP_RST_EXE), PT:=T#200MS);
grpResetEnd(IN:=(state=EStopSM.GRP_RST_END), PT:=T#200MS);


CASE state OF
	EStopSM.STARTUP:
		_TwinSafeGroup_Reset := TRUE;
		_TwinSafe_Run := TRUE;
		_resetGroup := FALSE;
		_switchName := '';
		_switchIdx := -1; //Emergency stop ok
		state := EStopSM.WAITRESET;
		
	EStopSM.WAITRESET:
		_TwinSafe_Run := TRUE;
		_TwinSafeGroup_Reset := FALSE;
		IF (NOT startUpTimer.Q) THEN
			state := EStopSM.GRP_RST_START;
		END_IF
	
	EStopSM.IDLE:
		_TwinSafe_Run := TRUE;
		_TwinSafeGroup_Reset := FALSE;
		IF (NOT _NoEStopDetected) AND Enabled THEN
			state := EStopSM.ESTOP;
		ELSIF _resetGroup THEN
			_resetGroup := FALSE;
			state := EStopSM.GRP_RST_START;
		END_IF
	
	EStopSM.ESTOP:
		_TwinSafe_Run := TRUE;
		_TwinSafeGroup_Reset := FALSE;
		IF _resetGroup THEN
			_resetGroup := FALSE;
			state := EStopSM.GRP_RST_START;
		ELSIF NOT _NoEStopDetected THEN
			_switchIdx := -1;
			// Find the first activated EStop switch 
			FOR _idx := 0 TO Parameters.SizeOfEStopArray-1 DO
				IF NOT _EStopSwitches[_idx] THEN
					_switchIdx := _idx;
					_switchName := Config.switchname[_idx];
					EXIT;
				END_IF
			END_FOR
		ELSE
			state := EStopSM.ESTOP_RELEASED;	
		END_IF
	
	EStopSM.ESTOP_RELEASED:
		_TwinSafe_Run := TRUE;
		_TwinSafeGroup_Reset := FALSE;
		_switchName := '';
		_switchIdx := -1;
		state := EStopSM.IDLE;
	
	ESTOPSM.GRP_RST_START:
		_TwinSafe_Run := FALSE;
		_TwinSafeGroup_Reset := FALSE;
		IF grpResetStart.Q THEN
			state := ESTOPSM.GRP_RST_EXE;
		END_IF
		
	ESTOPSM.GRP_RST_EXE:
		_TwinSafe_Run := FALSE;
		_TwinSafeGroup_Reset := TRUE;
		IF grpResetExe.Q THEN
			state := ESTOPSM.GRP_RST_END;
		END_IF

	ESTOPSM.GRP_RST_END:
		_TwinSafe_Run := FALSE;
		_TwinSafeGroup_Reset := FALSE;
		IF grpResetEnd.Q THEN
			state := ESTOPSM.IDLE;
		END_IF
END_CASE

{attribute 'monitoring' := 'call'}
{attribute 'TcRpcEnable'}
PROPERTY Activated : BOOL
GET
Activated := ((NOT _NoEStopDetected) OR _externEStop) AND Enabled;
END_GET
END_PROPERTY

{attribute 'monitoring' := 'call'}
{attribute 'TcRpcEnable'}
PROPERTY ActivatedSwitchIdx : INT
GET
ActivatedSwitchIdx := _switchIdx;
END_GET
END_PROPERTY

{attribute 'monitoring' := 'call'}
{attribute 'TcRpcEnable'}
PROPERTY ActivatedSwitchName : p7type.P6IdName
GET
ActivatedSwitchName := _switchName;
END_GET
END_PROPERTY

PROPERTY ExternEStop : BOOL
SET
_ExternEStop := ExternEStop;
END_SET
END_PROPERTY

{attribute 'monitoring' := 'call'}
{attribute 'TcRpcEnable'}
PROPERTY GroupError : BOOL
GET
GroupError := _TwinSafeGroupErrCom OR _TwinSafeGroupErrFB OR _TwinSafeGroupErrOther;
END_GET
END_PROPERTY

{attribute 'TcRpcEnable'}
METHOD resetGroupError : BOOL
_resetGroup := TRUE;
END_METHOD

END_FUNCTION_BLOCK

// TimingGenerators/SymmetricPulse
//Generates a pulse with 50% duty cycle
FUNCTION_BLOCK SymmetricPulse
VAR_INPUT
	CLK : TIME; // Time Period of signal. Signal is on CLK/2, and off CLK/2.
END_VAR
VAR_OUTPUT
END_VAR
VAR
	timer : TON;
	_value : BOOL;
END_VAR

timer(IN:=NOT timer.Q, PT:=CLK/2);
IF _value AND timer.Q THEN
	_value := FALSE;
ELSIF NOT _value AND timer.Q THEN
	_value := TRUE;
END_IF

PROPERTY Value : BOOL
GET
Value := _value;
END_GET
END_PROPERTY

END_FUNCTION_BLOCK

// EventManagement/AlarmAnalog
{attribute 'hide_all_locals'} 
FUNCTION_BLOCK ABSTRACT AlarmAnalog  EXTENDS AlarmEvent
VAR_INPUT
	LimitOn		: LREAL;
	LimitOff	: LREAL;
END_VAR
VAR
	_value		: LREAL;
	pipe		: SignalPipeline;
	distLimits	: LREAL;
END_VAR

_processing();

METHOD PROTECTED _createArguments : BOOL
SUPER^._createArguments();

THIS^.alarmEvt.ipArguments.AddLReal(_value);
END_METHOD

METHOD PROTECTED _processing : BOOL
VAR_INST
	state	: DINT;
	timerOn	: TON;
	timerOff: TON;
END_VAR
distLimits		:= LimitOn - LimitOff;

_processPipeline();

timerOn(IN:=  pipe.getBinaryValue(), PT:=T#1S);
timerOff(IN:=  NOT pipe.getBinaryValue(), PT:=T#1S);
			
CASE state OF
	0: 
		IF timerOn.Q THEN
			state := 1;
			THIS^.raise();
		END_IF
		
	1: 
		IF timerOff.Q THEN
			state := 0;
			THIS^.clear();
		END_IF 

	ELSE
		state := 0;
END_CASE
END_METHOD

METHOD ABSTRACT  _processPipeline : BOOL
END_METHOD

END_FUNCTION_BLOCK

// EventManagement/AlarmEvent
(* 
	This abstract class is the foundation for P6 Alarms.  Each  EventEntry in the Type System table has to include 
	a manual made ID. This ID is autogenerated but has to be modified according to the following describtion:
	
	Type of the ID is UDINT
	
	The hexadecimal representation is 6 siffre long and is shifted 8 bits to the left by an alarm. The positions are encoded as following

	DDDAAA##

	DDD represents a class of a device like winch or inverters. This gives a range of 4096 device classes
	AAA represents event class like high temperature. Example
	## is the numerical device id, which will be inserted when the instance for the alarm class is made
	
    16#00100201 would an alarm for a tripped inverter. DDD is 16#001 which represents the inverter classes while 
    AAA is 16#002 represents the high temperature alarm

	Parameter 0 is the Alarm Code
	Parameter 1 is the Dev ID
	Parameter 2 is the Dev Name
		
*)
{attribute 'hide'} 
{attribute 'hide_all_locals'}
FUNCTION_BLOCK ABSTRACT AlarmEvent
VAR_INPUT
	ID					: UDINT;
	IDName				: p7type.P6IDName;
END_VAR
VAR	
	alarmEvt			: FB_TCAlarm;
	sourceInfo			: FB_TCSourceInfo;	
	eventEntry			: TCEventEntry;
	createExstatus		: HRESULT;
END_VAR

METHOD PROTECTED _createArguments : BOOL
VAR
	alarmCode 		: UDINT;
END_VAR
THIS^.alarmEvt.ipArguments.Clear();

//  The EventId is put into the alarm definition in the type system. 
// The encoding of infomation into the EventId is documented in
// p7lib-basetypes/Events/Alarm Definitions.txt and in the Wiki  
alarmCode := SHL(THIS^.eventEntry.nEventId, 8) OR (THIS^.ID AND 16#FF);

THIS^.alarmEvt.ipArguments.AddUDInt(alarmCode);
THIS^.alarmEvt.ipArguments.AddUDInt(THIS^.ID);
THIS^.alarmEvt.ipArguments.AddString(THIS^.IDName);
END_METHOD

METHOD PROTECTED  _createEvent : BOOL
THIS^.sourceInfo.Clear();
THIS^.createExstatus := THIS^.alarmEvt.CreateEx(eventEntry, TRUE, THIS^.sourceInfo);
END_METHOD

{attribute 'TcRpcEnable'}
METHOD clear : BOOL
THIS^.alarmEvt.Clear(0, FALSE);
END_METHOD

{attribute 'TcRpcEnable'}
METHOD confirm : BOOL
THIS^.alarmEvt.Confirm(0);
END_METHOD

METHOD FB_init : BOOL
VAR_INPUT
	bInitRetains 	: BOOL; // if TRUE, the retain variables are initialized (warm start / cold start)
	bInCopyCode 	: BOOL;  // if TRUE, the instance afterwards gets moved into the copy code (online change)
	EventEntry		: TCEventEntry;
END_VAR
THIS^.eventEntry 	:= EventEntry;
THIS^._createEvent();
END_METHOD

{attribute 'TcRpcEnable'}
METHOD  raise : BOOL
THIS^._createArguments();
THIS^.alarmEvt.Raise(0);
END_METHOD

{attribute 'TcRpcEnable'}
PROPERTY Raised : BOOL
GET
Raised := THIS^.alarmEvt.bRaised;
END_GET
END_PROPERTY

END_FUNCTION_BLOCK

// EventManagement/AlarmAnalogValueHigh
(*
This class triggers an alarm, when a value is too high. A hysteresis is build in
*) 
{attribute 'hide_all_locals'}
FUNCTION_BLOCK AlarmAnalogValueHigh EXTENDS AlarmAnalog
VAR_INPUT
	Value		: LREAL;
END_VAR

_value := Value;
SUPER^();

METHOD _processPipeline : BOOL
THIS^.pipe
	.setLRealInput(THIS^.Value)
	.testGreaterOrEqual(Value := THIS^.limitOn - distLimits/2, Hysteresis := ABS(distLimits), MakeAnd := FALSE);
END_METHOD

END_FUNCTION_BLOCK

// EventManagement/AlarmAnalogValueLow
(*
This class triggers an alarm, when a value is too low. A hysteresis is build in
*) 
{attribute 'hide_all_locals'}
FUNCTION_BLOCK AlarmAnalogValueLow EXTENDS AlarmAnalog
VAR_INPUT
	Value	: LREAL;
END_VAR

_value := Value;
SUPER^();

METHOD _processPipeline : BOOL
THIS^.pipe
	.setLRealInput(THIS^.Value)
	.testLessOrEqual(Value := THIS^.limitOn - distLimits/2, Hysteresis := ABS(distLimits), MakeAnd := FALSE);
END_METHOD

END_FUNCTION_BLOCK

// EventManagement/AlarmCollector
{attribute 'hide_all_locals'}
FUNCTION_BLOCK AlarmCollector EXTENDS FB_ListenerBase2
VAR
	hr 						: HRESULT;
	criticalAlarmsRaised 	: DINT;
	warningAlarmsRaised 	: DINT;
	filter					: FB_TcEventFilter;
	started 				: BOOL;
	
	resettimer				: TOF;
	timeron					: BOOL;
	eventLogger				: FB_TcEventLogger;
	_confirmAlarms			: BOOL;
END_VAR

IF NOT started THEN
	Filter.Clear().IsAlarm();
			  	
	hr := THIS^.Subscribe2(Filter);
	started := TRUE;
ELSE
	update();
END_IF

{attribute 'TcRpcEnable'}
PROPERTY AlarmCritical : BOOL
GET
AlarmCritical :=  criticalAlarmsRaised > 0;
END_GET
END_PROPERTY

{attribute 'TcRpcEnable'}
PROPERTY AlarmWarning : BOOL
GET
AlarmWarning := warningAlarmsRaised > 0;
END_GET
END_PROPERTY

PROPERTY ConfirmAlarms : BOOL
SET
_confirmAlarms := ConfirmAlarms;
END_SET
END_PROPERTY

METHOD OnAlarmConfirmed : HRESULT
VAR_INPUT
	fbEvent : REFERENCE TO FB_TcEvent;
END_VAR
CASE fbEvent.eSeverity OF
	TCEventSeverity.Critical, TCEventSeverity.Error: 
		criticalAlarmsRaised := MAX(0, criticalAlarmsRaised - 1);
	ELSE 
		warningAlarmsRaised := MAX(0, warningAlarmsRaised - 1);
END_CASE

OnAlarmConfirmed := S_OK; // in order to receive more callbacks (Set <> S_OK in order to cancel the callbacks for this program cycle.)
END_METHOD

METHOD OnAlarmRaised : HRESULT
VAR_INPUT
	fbEvent : REFERENCE TO FB_TcEvent;
END_VAR
CASE fbEvent.eSeverity OF
	TCEventSeverity.Critical, TcEventSeverity.Error: 
		criticalAlarmsRaised := criticalAlarmsRaised + 1;
	ELSE 
		warningAlarmsRaised := warningAlarmsRaised + 1;
END_CASE


OnAlarmRaised := S_OK; // in order to receive more callbacks (Set <> S_OK in order to cancel the callbacks for this program cycle.)
END_METHOD

{attribute 'TcRpcEnable'}
METHOD reset : BOOL
timeron := TRUE;
END_METHOD

METHOD update : HRESULT
VAR_INST
	state : DINT;
END_VAR
resettimer(IN:= timeron, PT:=T#500MS);
IF resettimer.Q THEN
	criticalAlarmsRaised := 0;
	warningAlarmsRaised := 0;
	timeron := FALSE;
END_IF; 

CASE state OF
	0: 
		IF _confirmAlarms THEN
			state := 10;
		END_IF
		
	10:
		eventLogger.ConfirmAllAlarms(0);
		criticalAlarmsRaised := 0;
		warningAlarmsRaised := 0;
		state := 20;
 
	20:
		IF NOT _confirmAlarms THEN
			state := 0;	
		END_IF
END_CASE

update := SUPER^.Execute(); //retrieve events
END_METHOD

END_FUNCTION_BLOCK

// EventManagement/AlarmCollectorEx
FUNCTION_BLOCK AlarmCollectorEx EXTENDS FB_ListenerBase2
VAR CONSTANT
	TABLELEN : DINT := 40;
END_VAR
VAR_INPUT
	tableHMI 				: REFERENCE TO ARRAY[0..TABLELEN-1] OF AlarmTable;
END_VAR
VAR
	table 					: ARRAY[0..TABLELEN-1] OF EventProcessing;
	eventLogger				:  FB_TcEventLogger;
	filter					: FB_TcEventFilter;
	reqText 				: ARRAY[0..TABLELEN-1] OF FB_RequestEventText;
	
	systemtime				: TIMESTRUCT;
	criticalAlarmsRaised 	: DINT;
	warningAlarmsRaised 	: DINT;
	started 				: BOOL;
	
	resettimer				: TOF;
	timeron					: BOOL;
	plcTime					: STRING;
	_confirmAlarms			: BOOL;
	state					: DINT;
END_VAR

IF NOT started THEN
	Filter.Clear().IsAlarm();  	
	THIS^.Subscribe2(Filter);
	started := TRUE;
ELSE
	CASE state OF
		0: 
			IF _confirmAlarms THEN
				state := 10;
			END_IF
			
		10:
			eventLogger.ConfirmAllAlarms(0);
			criticalAlarmsRaised := 0;
			warningAlarmsRaised := 0;
			state := 20;
	 
		20:
			IF NOT _confirmAlarms THEN
				state := 0;	
			END_IF
	END_CASE
	
	this^.Execute();
END_IF

{attribute 'TcRpcEnable'}
PROPERTY AlarmCritical : BOOL
GET
AlarmCritical :=  criticalAlarmsRaised > 0;
END_GET
END_PROPERTY

{attribute 'TcRpcEnable'}
PROPERTY AlarmWarning : BOOL
GET
AlarmWarning := warningAlarmsRaised > 0;
END_GET
END_PROPERTY

PROPERTY ConfirmAlarms : BOOL
SET
_confirmAlarms := ConfirmAlarms;
END_SET
END_PROPERTY

METHOD PRIVATE copyTableToHMI : BOOL
VAR
	N : DINT;
	P : DINT;
END_VAR
P := 0;
FOR N := 0 TO TABLELEN-1 DO
	IF NOT __ISVALIDREF(THIS^.table[N].event) THEN
		CONTINUE;
	END_IF
	tableHMI[P].message := table[N].message;
	tableHMI[P].timestamp := table[N].timestamp; 
	tableHMI[P].eventID := table[N].eventID;
	P := P + 1; 
END_FOR

FOR N := P TO TABLELEN-1 DO
	tableHMI[N].message := '';
	tableHMI[N].timestamp := '';
	tableHMI[N].eventID := 0;
END_FOR
END_METHOD

METHOD PRIVATE delEvent : BOOL
VAR_INPUT
	event : REFERENCE TO FB_TcEvent;
END_VAR
VAR
	N : DINT;
END_VAR


FOR N := 0 TO TABLELEN-1 DO
	IF NOT __ISVALIDREF(table[N].event) THEN
		CONTINUE;
	END_IF 
	IF table[N].uid = event.nUniqueId THEN
		table[N].event REF= 0;
		EXIT;
	END_IF
END_FOR
copyTableToHMI();
END_METHOD

METHOD Execute : HRESULT
VAR_INST
	timelocal : FB_LocalSystemTime;
	msg : STRING(255);
	res : BOOL;
	b  : BOOL;
	e : BOOL;
END_VAR
Execute := SUPER^.Execute(); //retrieve events

resettimer(IN:= timeron, PT:=T#500MS);
IF resettimer.Q THEN
	criticalAlarmsRaised := 0;
	warningAlarmsRaised := 0;
	timeron := FALSE;
END_IF; 

timelocal(
	sNetId 			:= '',
	bEnable 		:= TRUE,
	dwCycle			:= 10,
	dwOpt			:= 0,
	tTimeOut		:= T#10S,
	systemtime 		=> systemtime
);	


getText();
END_METHOD

METHOD PRIVATE getText : BOOL
VAR_INST
	msg : STRING(255);
	N : DINT;
END_VAR
FOR N := 0 TO TABLELEN-1 DO
	IF NOT __ISVALIDREF(table[N].event) THEN
		CONTINUE;
	END_IF 
	IF (NOT table[N].hasTxt) THEN
		IF (NOT reqText[N].bBusy) AND (NOT reqText[N].bError ) THEN
			reqText[N].GetString(msg, SIZEOF(msg));	
			table[N].message := msg;
			table[N].hasTxt := TRUE;		
		END_IF
		copyTableToHMI();
	END_IF
END_FOR
END_METHOD

METHOD PRIVATE insertEvent : BOOL
VAR_INPUT
	event : REFERENCE TO FB_TcEvent;
END_VAR
VAR_INST
	N 		: DINT;
	msg : STRING(255);
	res : BOOL;
END_VAR
plcTime := SYSTEMTIME_TO_STRING(systemtime);

FOR N := 0 TO TABLELEN-1 DO
	IF NOT __ISVALIDREF(table[N].event) THEN
		table[N].message := 'Error ALARMTEXT';
		table[N].event REF= event;
		table[N].uid := event.nUniqueId;
		
		table[N].eventID := event.nEventId;
		table[N].timestamp := plcTime;
		table[N].hasTxt := FALSE;
		
		reqText[N].Request(eventClass:=Event.EventClass, nEventId:=Event.nEventId, nLangId:=1033, ipArgs:=Event.ipArguments );
		EXIT;
	END_IF
END_FOR
END_METHOD

METHOD OnAlarmCleared : HRESULT
VAR_INPUT
	fbEvent : REFERENCE TO FB_TcEvent;
END_VAR

delEvent(fbEvent);
OnAlarmCleared := S_OK;
END_METHOD

METHOD OnAlarmConfirmed : HRESULT
VAR_INPUT
	fbEvent : REFERENCE TO FB_TcEvent;
END_VAR
VAR 
	a:INT;
END_VAR
CASE fbEvent.eSeverity OF
	TCEventSeverity.Critical: 
		criticalAlarmsRaised := MAX(0,criticalAlarmsRaised) - 1;
	ELSE 
		warningAlarmsRaised := MAX(0, warningAlarmsRaised - 1);
END_CASE

OnAlarmConfirmed := S_OK; // in order to receive more callbacks (Set <> S_OK in order to cancel the callbacks for this program cycle.)
END_METHOD

METHOD OnAlarmRaised : HRESULT
VAR_INPUT
	fbEvent : REFERENCE TO FB_TcEvent;
END_VAR
VAR
	b : BOOL;
	m : String(80);
END_VAR
CASE fbEvent.eSeverity OF
	TCEventSeverity.Critical: 
		criticalAlarmsRaised := criticalAlarmsRaised + 1;
	ELSE 
		warningAlarmsRaised := warningAlarmsRaised + 1;
END_CASE

insertEvent(fbEvent);

//queryMsg.Request(eventClass:=fbEvent.EventClass, nEventId:=fbEvent.nEventId, nLangId:=1031, ipArgs:=fbEvent.ipArguments );

OnAlarmRaised := S_OK; // in order to receive more callbacks (Set <> S_OK in order to cancel the callbacks for this program cycle.)
END_METHOD

{attribute 'TcRpcEnable'}
METHOD reset : BOOL
timeron := TRUE;
END_METHOD

END_FUNCTION_BLOCK

// EventManagement/AlarmDigital
{attribute 'hide_all_locals'}
FUNCTION_BLOCK AlarmDigital EXTENDS AlarmEvent
VAR_INPUT
	Value		: BOOL;
	TimeSpan 	: TIME;
END_VAR
VAR
	timer	 	: TON;
	minTime		: TOF;
	state    	: DINT;
END_VAR

SUPER^();

timer(IN:= Value, PT:= THIS^.TimeSpan);
minTime(IN:=timer.Q, PT:=T#1S);

CASE state OF
	0: 
		IF minTime.Q THEN
			THIS^.raise();
			state := 1;
		END_IF
		
	1:
		IF NOT minTime.Q THEN
			THIS^.clear();
			state := 0;
		END_IF
 
	ELSE
		state := 0;
END_CASE

END_FUNCTION_BLOCK

// EventManagement/AlarmDigitalEx
{attribute 'hide_all_locals'}
FUNCTION_BLOCK AlarmDigitalEx EXTENDS AlarmEvent
VAR_INPUT
	Value		: BOOL;
	TimeSpan 	: TIME;
	ValueAnalog	: LREAL;
END_VAR
VAR
	timer	 	: TON;
	state    	: DINT;
END_VAR

SUPER^();

timer(IN:= Value, PT:= THIS^.TimeSpan);

CASE state OF
	0: 
		IF timer.Q THEN
			THIS^.raise();
			state := 1;
		END_IF
		
	1:
		IF NOT timer.Q THEN
			THIS^.clear();
			state := 0;
		END_IF
 
	ELSE
		state := 0;
END_CASE

METHOD PROTECTED _createArguments : BOOL
SUPER^._createArguments();

THIS^.alarmEvt.ipArguments.AddLReal(ValueAnalog);
END_METHOD

END_FUNCTION_BLOCK

// EventManagement/AlarmOilFilter
{attribute 'hide_all_locals'}
FUNCTION_BLOCK AlarmOilFilter EXTENDS AlarmEvent
VAR_INPUT
	SensorFilter		: IAnalogSensor;
	SensorTemperature	: IAnalogSensor;	
	TemperatureMin		: LREAL;
END_VAR
VAR
	state				: DINT;
	timer				: TON;
END_VAR

SUPER^();

timer(IN:= (sensorFilter.Value > 0.5) AND (sensorTemperature.Value > TemperatureMin), PT:=T#1S);


CASE state OF
	0: 
		IF timer.Q THEN
			state := 1;
			THIS^.raise();
		END_IF
		
	1: 
		IF NOT timer.Q THEN
			THIS^.clear();
			state := 0;
		END_IF
		
	ELSE
		state := 0;
END_CASE

END_FUNCTION_BLOCK

// EventManagement/AlarmSensorError
{attribute 'hide_all_locals'}
FUNCTION_BLOCK AlarmSensorError EXTENDS AlarmEvent
VAR_INPUT
	Sensor : IAnalogSensor;
END_VAR
VAR
	timer	 : TON;
	state    : DINT;	
END_VAR

SUPER^();

timer(IN:= Sensor.Error, PT:= T#0.1S);

CASE state OF
	0: 
		IF timer.Q THEN
			state := 1;
			THIS^.raise();
		END_IF
		
	1: 
		IF NOT timer.Q THEN
			state := 0;
			THIS^.clear();
		END_IF 
	ELSE
		state := 0;
END_CASE

END_FUNCTION_BLOCK

// EventManagement/AlarmSensorValueHigh
{attribute 'hide_all_locals'}
FUNCTION_BLOCK AlarmSensorValueHigh EXTENDS AlarmAnalog
VAR_INPUT	
	Sensor	: IAnalogSensor;
END_VAR

_value := Sensor.Value;
SUPER^();

METHOD _processPipeline : BOOL
THIS^.pipe
	.setLRealInput(_value)
	.testGreaterOrEqual(Value := THIS^.limitOn - distLimits/2, Hysteresis := ABS(distLimits), MakeAnd := FALSE);
END_METHOD

END_FUNCTION_BLOCK

// EventManagement/AlarmSensorValueLow
{attribute 'hide_all_locals'}
FUNCTION_BLOCK AlarmSensorValueLow EXTENDS AlarmAnalog
VAR_INPUT	
	Sensor	: IAnalogSensor;
END_VAR

_value := Sensor.Value;
SUPER^();

METHOD _processPipeline : BOOL
THIS^.pipe
	.setLRealInput(_value)
	.testLessOrEqual(Value := THIS^.limitOn - distLimits/2, Hysteresis := ABS(distLimits), MakeAnd := FALSE);
END_METHOD

END_FUNCTION_BLOCK

// EventManagement/AlarmSimple
{attribute 'hide_all_locals'}
FUNCTION_BLOCK AlarmSimple EXTENDS AlarmEvent

SUPER^();

END_FUNCTION_BLOCK

// EventManagement/StartupDelay
FUNCTION_BLOCK StartupDelay
VAR
	delayTime 	: TIME;
	timer 		: TON; 
END_VAR

timer(IN := TRUE, PT:=delayTime);

PROPERTY Done : BOOL
GET
Done := timer.Q;
END_GET
END_PROPERTY

METHOD FB_init : BOOL
VAR_INPUT
	bInitRetains : BOOL; // if TRUE, the retain variables are initialized (warm start / cold start)
	bInCopyCode : BOOL;  // if TRUE, the instance afterwards gets moved into the copy code (online change)
	delayTime : TIME;
END_VAR
THIS^.delayTime := delayTime;
END_METHOD

END_FUNCTION_BLOCK

// Fieldbus/Ethercat
(*
Purpose
=======
This class is providing functionality to implement CoE queries for Ethercat devices. Each request needs it's 
own instance to avoid problems with concurrency.  

Caveats
=======
All functions are a sort of asynchronous, which means they returning busy until the result was returned from 
Twincat. 

Methods And Properties
======================
*)
{attribute 'no_explicit_call' := 'do not call this POU directly'} 
{attribute 'hide_all_locals'}
FUNCTION_BLOCK Ethercat
VAR CONSTANT
	_objectIdentity : EthercatCoEObjectArray := [
		(para:= 101801, idx:= 16#1018, sidx:= 16#01, tclass:= EthTypes.TDWORD),	// Vendor ID
		(para:= 101802, idx:= 16#1018, sidx:= 16#02, tclass:= EthTypes.TDWORD),	// Product Code
		(para:= 101803, idx:= 16#1018, sidx:= 16#03, tclass:= EthTypes.TDWORD),	// Revision
		(para:= 16#FFFF_FFFF, idx:= 16#0000, sidx:= 16#00, tclass:= EthTypes.TWORD) // EoL
	];
	
END_VAR
VAR
	_objValueIdentity :  EthercatCoEValueArray;
END_VAR

(*
Purpose
=======

This function is reading any data object via SDO.
*)
METHOD PRIVATE _readCoEData : EFieldbusQueryResult
VAR_INPUT CONSTANT 
	AMSAddr				: AMSADDR;	
END_VAR
VAR_INPUT
	Index				: UINT;
	SubIndex			: BYTE;
	BufferPointer		: PVOID;
	BufferLen			: UDINT;
END_VAR
VAR_INST
	DataReader 			: FB_EcCoESDORead;
	state 				: ESimpleFieldbusSM;
	doRun				: BOOL; 	
	busy				: BOOL;
	error				: BOOL;
	result 				: EFieldbusQueryResult;		
	nErrId				: UDINT;
END_VAR
DataReader(
	sNetId 					:= F_CreateAMSNetID(AMSAddr.netId),
	nSlaveAddr				:= AMSAddr.port,
	nIndex					:= Index,
	nSubIndex				:= SubIndex,
	pDstBuf					:= BufferPointer,
	cbBufLen				:= BufferLen,
	bExecute				:= doRun,
	tTimeout				:= T#500MS,
	bBusy					=> busy,
	bError 					=> error,
	nErrId 					=> nErrId);


CASE state OF
	ESimpleFieldbusSM.IDLE:
		doRun 	:= FALSE; 
		result 	:= EFieldbusQueryResult.BUSY;
		state 	:= ESimpleFieldbusSM.STARTUP;
		
	ESimpleFieldbusSM.STARTUP: 
		doRun 	:= TRUE; 
		result 	:= EFieldbusQueryResult.BUSY;
		state 	:= ESimpleFieldbusSM.WAITONRESULT;

	ESimpleFieldbusSM.WAITONRESULT: 
		doRun 	:= TRUE; 
		result 	:= EFieldbusQueryResult.BUSY;
		IF (NOT busy) OR error THEN
			state 	:= ESimpleFieldbusSM.RESULT;
		END_IF;
		
	ESimpleFieldbusSM.RESULT: 
		doRun 	:= FALSE; 
		IF error THEN
			result 	:= EFieldbusQueryResult.FAIL;
		ELSE
			result 	:= EFieldbusQueryResult.OK;
		END_IF
		state 	:= ESimpleFieldbusSM.STARTUP;
END_CASE

_readCoEData := result;
END_METHOD

METHOD PRIVATE _writeCoEData : EFieldbusQueryResult
VAR_INPUT CONSTANT
	AMSAddr				: AMSADDR;	
END_VAR
VAR_INPUT
	Index				: UINT;
	SubIndex			: BYTE;
	BufferPointer		: PVOID;
	BufferLen			: UDINT;
END_VAR
VAR_INST
	DataWriter 			: FB_EcCoESdoWrite;
	state 				: ESimpleFieldbusSM;
	doRun				: BOOL; 	
	busy				: BOOL;
	error				: BOOL;
	result 				: EFieldbusQueryResult;		
	nErrId				: UDINT;
END_VAR
DataWriter(
	sNetId 					:= F_CreateAMSNetID(AMSAddr.netId),
	nSlaveAddr				:= AMSAddr.port,
	nIndex					:= Index,
	nSubIndex				:= SubIndex,
	pSrcBuf					:= BufferPointer,
	cbBufLen				:= BufferLen,
	bExecute				:= doRun,
	tTimeout				:= T#500MS,
	bBusy					=> busy,
	bError 					=> error,
	nErrId 					=> nErrId);


CASE state OF
	ESimpleFieldbusSM.IDLE:
		doRun 	:= FALSE; 
		result 	:= EFieldbusQueryResult.BUSY;
		state 	:= ESimpleFieldbusSM.STARTUP;
		
	ESimpleFieldbusSM.STARTUP: 
		doRun 	:= TRUE; 
		result 	:= EFieldbusQueryResult.BUSY;
		state 	:= ESimpleFieldbusSM.WAITONRESULT;

	ESimpleFieldbusSM.WAITONRESULT: 
		doRun 	:= TRUE; 
		result 	:= EFieldbusQueryResult.BUSY;
		IF (NOT busy) OR error THEN
			state 	:= ESimpleFieldbusSM.RESULT;
		END_IF;
		
	ESimpleFieldbusSM.RESULT: 
		doRun 	:= FALSE; 
		IF error THEN
			result 	:= EFieldbusQueryResult.FAIL;
		ELSE
			result 	:= EFieldbusQueryResult.OK;
		END_IF
		state 	:= ESimpleFieldbusSM.STARTUP;
END_CASE

_writeCoEData := result;
END_METHOD

METHOD isDevice : EFieldbusQueryResult
VAR_INPUT CONSTANT
	AMSAddr			: AMSADDR;
END_VAR
VAR_INPUT
	VendorID		: DWORD;
	ProductCode		: DWORD;
	Revision		: DWORD; // optional. When 0 Revision is ignored
	Exec			: BOOL;
	Index 			: REFERENCE TO DINT := 0;
END_VAR
VAR_INST
	result			: EFieldbusQueryResult;
	trigger			: R_TRIG;
	state			: INT;
	execRead		: BOOL;
END_VAR

result := readCoEValueArray(AMSAddr, ADR(_objectIdentity), ADR(_objValueIdentity), state = 10, Index);


CASE state OF 
	0: 
		isDevice := EFieldbusQueryResult.BUSY;
		IF Exec THEN
			state := 10;
		END_IF
		
	10:
		isDevice := EFieldbusQueryResult.BUSY;
		IF result <> EFieldbusQueryResult.BUSY THEN
			state := 20;
		END_IF
		
	20:
		IF result = EFieldbusQueryResult.OK THEN
			IF Revision <> 0 THEN
				IF VendorID = _objValueIdentity[0].VDWORD AND 
					ProductCode = _objValueIdentity[1].VDWORD THEN
					isDevice := EFieldbusQueryResult.OK;
				ELSE
					isDevice := EFieldbusQueryResult.FAIL;
				END_IF
			END_IF
		ELSE
			isDevice := EFieldbusQueryResult.FAIL;
		END_IF
		state := 30;
		
	30:
		IF NOT Exec THEN
			state := 0;			
		END_IF
END_CASE
END_METHOD

(*
Purpose
=======

This function is reading a byte object via SDO.

*)
METHOD readCoEDataBYTE : EFieldbusQueryResult
VAR_INPUT CONSTANT
	AMSAddr				: AMSADDR;	
END_VAR
VAR_INPUT
	Index				: UINT;
	SubIndex			: BYTE;
	Value 				: REFERENCE TO BYTE;
END_VAR

readCoEDataBYTE := _readCoEData(AMSAddr, Index, SubIndex, ADR(Value), SIZEOF(Value));
END_METHOD

(*
Purpose
=======

This function is reading a dint object via SDO.

*)
METHOD readCoEDataDINT : EFieldbusQueryResult
VAR_INPUT CONSTANT
	AMSAddr				: AMSADDR;	
END_VAR
VAR_INPUT
	Index				: UINT;
	SubIndex			: BYTE;
	Value 				: REFERENCE TO DINT;
END_VAR

readCoEDataDINT := _readCoEData(AMSAddr, Index, SubIndex, ADR(Value), SIZEOF(Value));
END_METHOD

(*
Purpose
=======

This function is reading a dword object via SDO.

*)
METHOD readCoEDataDWORD : EFieldbusQueryResult
VAR_INPUT CONSTANT
	AMSAddr				: AMSADDR;	
END_VAR
VAR_INPUT
	Index				: UINT;
	SubIndex			: BYTE;
	Value 				: REFERENCE TO DWORD;
END_VAR

readCoEDataDWORD := _readCoEData(AMSAddr, Index, SubIndex, ADR(Value), SIZEOF(Value));
END_METHOD

(*
Purpose
=======

This function is reading a int object via SDO.

*)
METHOD readCoEDataINT : EFieldbusQueryResult
VAR_INPUT CONSTANT
	AMSAddr				: AMSADDR;	
END_VAR
VAR_INPUT
	Index				: UINT;
	SubIndex			: BYTE;
	Value 				: REFERENCE TO INT;
END_VAR

readCoEDataINT := _readCoEData(AMSAddr, Index, SubIndex, ADR(Value), SIZEOF(Value));
END_METHOD

(*
Purpose
=======

This function is reading a lint object via SDO.

*)
METHOD readCoEDataLINT : EFieldbusQueryResult
VAR_INPUT CONSTANT
	AMSAddr				: AMSADDR;	
END_VAR
VAR_INPUT
	Index				: UINT;
	SubIndex			: BYTE;
	Value 				: REFERENCE TO LINT;
END_VAR

readCoEDataLINT := _readCoEData(AMSAddr, Index, SubIndex, ADR(Value), SIZEOF(Value));
END_METHOD

(*
Purpose
=======

This function is reading a lreal object via SDO.

*)
METHOD readCoEDataLREAL : EFieldbusQueryResult
VAR_INPUT CONSTANT
	AMSAddr				: AMSADDR;	
END_VAR
VAR_INPUT
	Index				: UINT;
	SubIndex			: BYTE;
	Value 				: REFERENCE TO LREAL;
END_VAR

readCoEDataLREAL := _readCoEData(AMSAddr, Index, SubIndex, ADR(Value), SIZEOF(Value));
END_METHOD

(*
Purpose
=======

This function is reading a lword object via SDO.

*)
METHOD readCoEDataLWORD : EFieldbusQueryResult
VAR_INPUT CONSTANT
	AMSAddr				: AMSADDR;	
END_VAR
VAR_INPUT
	Index				: UINT;
	SubIndex			: BYTE;
	Value 				: REFERENCE TO LWORD;
END_VAR

readCoEDataLWORD := _readCoEData(AMSAddr, Index, SubIndex, ADR(Value), SIZEOF(Value));
END_METHOD

(*
Purpose
=======

This function is reading a real object via SDO.

*)
METHOD readCoEDataREAL : EFieldbusQueryResult
VAR_INPUT CONSTANT
	AMSAddr				: AMSADDR;	
END_VAR
VAR_INPUT
	Index				: UINT;
	SubIndex			: BYTE;
	Value 				: REFERENCE TO REAL;
END_VAR

readCoEDataREAL := _readCoEData(AMSAddr, Index, SubIndex, ADR(Value), SIZEOF(Value));
END_METHOD

(*
Purpose
=======

This function is reading a sint object via SDO.

*)
METHOD readCoEDataSINT : EFieldbusQueryResult
VAR_INPUT CONSTANT
	AMSAddr				: AMSADDR;	
END_VAR
VAR_INPUT
	Index				: UINT;
	SubIndex			: BYTE;
	Value 				: REFERENCE TO SINT;
END_VAR

readCoEDataSINT := _readCoEData(AMSAddr, Index, SubIndex, ADR(Value), SIZEOF(Value));
END_METHOD

(*
Purpose
=======

This function is reading a uint object via SDO.

*)
METHOD readCoEDataUDINT : EFieldbusQueryResult
VAR_INPUT CONSTANT
	AMSAddr				: AMSADDR;	
END_VAR
VAR_INPUT
	Index				: UINT;
	SubIndex			: BYTE;
	Value 				: REFERENCE TO UDINT;
END_VAR

readCoEDataUDINT := _readCoEData(AMSAddr, Index, SubIndex, ADR(Value), SIZEOF(Value));
END_METHOD

(*
Purpose
=======

This function is reading a uint object via SDO.

*)
METHOD readCoEDataUINT : EFieldbusQueryResult
VAR_INPUT CONSTANT
	AMSAddr				: AMSADDR;	
END_VAR
VAR_INPUT
	Index				: UINT;
	SubIndex			: BYTE;
	Value 				: REFERENCE TO UINT;
END_VAR

readCoEDataUINT := _readCoEData(AMSAddr, Index, SubIndex, ADR(Value), SIZEOF(Value));
END_METHOD

(*
Purpose
=======

This function is reading a ulint object via SDO.

*)
METHOD readCoEDataULINT : EFieldbusQueryResult
VAR_INPUT CONSTANT
	AMSAddr				: AMSADDR;	
END_VAR
VAR_INPUT
	Index				: UINT;
	SubIndex			: BYTE;
	Value 				: REFERENCE TO ULINT;
END_VAR

readCoEDataULINT := _readCoEData(AMSAddr, Index, SubIndex, ADR(Value), SIZEOF(Value));
END_METHOD

(*
Purpose
=======

This function is reading a usint object via SDO.

*)
METHOD readCoEDataUSINT : EFieldbusQueryResult
VAR_INPUT CONSTANT
	AMSAddr				: AMSADDR;	
END_VAR
VAR_INPUT
	Index				: UINT;
	SubIndex			: BYTE;
	Value 				: REFERENCE TO USINT;
END_VAR

readCoEDataUSINT := _readCoEData(AMSAddr, Index, SubIndex, ADR(Value), SIZEOF(Value));
END_METHOD

(*
Purpose
=======

This function is reading a word object via SDO.

*)
METHOD readCoEDataWORD : EFieldbusQueryResult
VAR_INPUT CONSTANT
	AMSAddr				: AMSADDR;	
END_VAR
VAR_INPUT
	Index				: UINT;
	SubIndex			: BYTE;
	Value 				: REFERENCE TO WORD;
END_VAR

readCoEDataWORD := _readCoEData(AMSAddr, Index, SubIndex, ADR(Value), SIZEOF(Value));
END_METHOD

METHOD readCoEValueArray : EFieldbusQueryResult
VAR_INPUT CONSTANT
	AMSAddr			: AMSADDR;
	Objects			: POINTER TO EthercatCoEObjectArray;	
	Values 			: POINTER TO EthercatCoEValueArray; 	
END_VAR
VAR_INPUT
	Exec			: BOOL;
	Index			: REFERENCE TO DINT := 0;	
END_VAR
VAR_INST
	state			: EthWriteCoEArraySM;
	N 				: DINT;
	result			: EFieldbusQueryResult;
	trigger			: R_TRIG;
	w : DWORD;
END_VAR
trigger(CLK:=Exec);

IF NOT Exec THEN
	state := 0;
END_IF

CASE state OF
	EthWriteCoEArraySM.IDLE: 	
		readCoEValueArray := EFieldbusQueryResult.BUSY;
		IF trigger.Q THEN
			state := EthWriteCoEArraySM.INCR;
			N := -1;
		END_IF
		
	EthWriteCoEArraySM.WRITE: 
		readCoEValueArray := EFieldbusQueryResult.BUSY;
		CASE Objects^[N].tclass OF
			EthTypes.TBYTE:
				result := readCoEDataBYTE(AMSAddr, Objects^[N].idx, Objects^[N].sidx, Values^[N].VBYTE);
			EthTypes.TWORD:
				result := readCoEDataWORD(AMSAddr, Objects^[N].idx, Objects^[N].sidx, Values^[N].VWORD);
			EthTypes.TDWORD:
				result := readCoEDataDWORD(AMSAddr, Objects^[N].idx, Objects^[N].sidx, Values^[N].VDWORD);
			EthTypes.TLWORD:
				result := readCoEDataLWORD(AMSAddr, Objects^[N].idx, Objects^[N].sidx, Values^[N].VLWORD);
			EthTypes.TSINT:
				result := readCoEDataSINT(AMSAddr, Objects^[N].idx, Objects^[N].sidx, Values^[N].VSINT);
			EthTypes.TUSINT:
				result := readCoEDataUSINT(AMSAddr, Objects^[N].idx, Objects^[N].sidx, Values^[N].VUSINT);
			EthTypes.TINT:
				result := readCoEDataINT(AMSAddr, Objects^[N].idx, Objects^[N].sidx, Values^[N].VINT);
			EthTypes.TUINT:
				result := readCoEDataUINT(AMSAddr, Objects^[N].idx, Objects^[N].sidx, Values^[N].VUINT);
			EthTypes.TDINT:
				result := readCoEDataDINT(AMSAddr, Objects^[N].idx, Objects^[N].sidx, Values^[N].VDINT);
			EthTypes.TUDINT:
				result := readCoEDataUDINT(AMSAddr, Objects^[N].idx, Objects^[N].sidx, Values^[N].VUDINT);
			EthTypes.TLINT:
				result := readCoEDataLINT(AMSAddr, Objects^[N].idx, Objects^[N].sidx, Values^[N].VLINT);
			EthTypes.TULINT:
				result := readCoEDataULINT(AMSAddr, Objects^[N].idx, Objects^[N].sidx, Values^[N].VULINT);
			EthTypes.TREAL:
				result := readCoEDataREAL(AMSAddr, Objects^[N].idx, Objects^[N].sidx, Values^[N].VREAL);
			EthTypes.TLREAL:
				result := readCoEDataLREAL(AMSAddr, Objects^[N].idx, Objects^[N].sidx, Values^[N].VLREAL);
		END_CASE

		IF __ISVALIDREF(Index) THEN
			Index := N;
		END_IF

		CASE result OF
			EFieldbusQueryResult.FAIL:
				state := EthWriteCoEArraySM.ERROR;
			EFieldbusQueryResult.OK:
				state := EthWriteCoEArraySM.INCR;				
		END_CASE
	
	EthWriteCoEArraySM.INCR:
		readCoEValueArray := EFieldbusQueryResult.BUSY;
		N := N + 1;
		IF N > Parameters.SizeOfEthCoEValues-1 OR Objects^[N].para = 16#FFFF_FFFF THEN
			state := EthWriteCoEArraySM.READY;
		ELSE
			state := EthWriteCoEArraySM.WRITE;
		END_IF
		
	EthWriteCoEArraySM.READY:
		readCoEValueArray := EFieldbusQueryResult.OK;
		IF NOT Exec THEN
			state := EthWriteCoEArraySM.IDLE;
		END_IF

	EthWriteCoEArraySM.ERROR:		
		readCoEValueArray := EFieldbusQueryResult.FAIL;
		IF NOT Exec THEN
			state := EthWriteCoEArraySM.IDLE;
		END_IF		
		
END_CASE
END_METHOD

METHOD wait : EFieldbusQueryResult
VAR_INPUT
	WaitingTime 		: TIME; 
	Exec				: BOOL;
END_VAR
VAR_INST
	timer				: TON;
	state 				: ESimpleFieldbusSM;
	doRun				: BOOL; 	
	busy				: BOOL;
	result 				: EFieldbusQueryResult;			
END_VAR
timer(IN:=state=ESimpleFieldbusSM.WAITONRESULT, PT:=WaitingTime);

CASE state OF
	ESimpleFieldbusSM.IDLE: 	
		wait := EFieldbusQueryResult.BUSY;
		IF Exec THEN
			state := ESimpleFieldbusSM.WAITONRESULT;
		END_IF
		
	ESimpleFieldbusSM.WAITONRESULT: 
		wait := EFieldbusQueryResult.BUSY;
		IF timer.Q THEN
			state := ESimpleFieldbusSM.RESULT;						
		END_IF

	ESimpleFieldbusSM.RESULT: 
		wait := EFieldbusQueryResult.OK;
		IF NOT Exec THEN
			state := ESimpleFieldbusSM.IDLE;
		END_IF
END_CASE
END_METHOD

(*
Purpose
=======

This function is writing a byte object via SDO.

*)
METHOD writeCoEDataBYTE : EFieldbusQueryResult
VAR_INPUT
	AMSAddr				: AMSAddr;
	Index				: UINT;
	SubIndex			: BYTE;
	Value 				: BYTE;
END_VAR

writeCoEDataBYTE := _writeCoEData(AMSAddr, Index, SubIndex, ADR(Value), SIZEOF(Value));
END_METHOD

(*
Purpose
=======

This function is writing a dint object via SDO.

*)
METHOD writeCoEDataDINT : EFieldbusQueryResult
VAR_INPUT CONSTANT
	AMSAddr				: AMSADDR;	
END_VAR
VAR_INPUT
	Index				: UINT;
	SubIndex			: BYTE;
	Value 				: DINT;
END_VAR

writeCoEDataDINT := _writeCoEData(AMSAddr, Index, SubIndex, ADR(Value), SIZEOF(Value));
END_METHOD

(*
Purpose
=======

This function is writing a dword object via SDO.

*)
METHOD writeCoEDataDWORD : EFieldbusQueryResult
VAR_INPUT CONSTANT
	AMSAddr				: AMSADDR;	
END_VAR
VAR_INPUT
	Index				: UINT;
	SubIndex			: BYTE;
	Value 				: DWORD;
END_VAR

writeCoEDataDWORD := _writeCoEData(AMSAddr, Index, SubIndex, ADR(Value), SIZEOF(Value));
END_METHOD

(*
Purpose
=======

This function is writing a uint object via SDO.
*)
METHOD writeCoEDataINT : EFieldbusQueryResult
VAR_INPUT CONSTANT
	AMSAddr				: AMSADDR;	
END_VAR
VAR_INPUT
	Index				: UINT;
	SubIndex			: BYTE;
	Value 				: INT;
END_VAR

writeCoEDataINT := _writeCoEData(AMSAddr, Index, SubIndex, ADR(Value), SIZEOF(Value));
END_METHOD

(*
Purpose
=======

This function is writing a lint object via SDO.

*)
METHOD writeCoEDataLINT : EFieldbusQueryResult
VAR_INPUT CONSTANT
	AMSAddr				: AMSADDR;	
END_VAR
VAR_INPUT
	Index				: UINT;
	SubIndex			: BYTE;
	Value 				: LINT;
END_VAR

writeCoEDataLINT := _writeCoEData(AMSAddr, Index, SubIndex, ADR(Value), SIZEOF(Value));
END_METHOD

(*
Purpose
=======

This function is writing a lreal object via SDO.

*)
METHOD writeCoEDataLREAL : EFieldbusQueryResult
VAR_INPUT CONSTANT
	AMSAddr				: AMSADDR;	
END_VAR
VAR_INPUT
	Index				: UINT;
	SubIndex			: BYTE;
	Value 				: LREAL;
END_VAR

writeCoEDataLREAL := _writeCoEData(AMSAddr, Index, SubIndex, ADR(Value), SIZEOF(Value));
END_METHOD

(*
Purpose
=======

This function is writing a lword object via SDO.

*)
METHOD writeCoEDataLWORD : EFieldbusQueryResult
VAR_INPUT CONSTANT
	AMSAddr				: AMSADDR;	
END_VAR
VAR_INPUT
	Index				: UINT;
	SubIndex			: BYTE;
	Value 				: LWORD;
END_VAR

writeCoEDataLWORD := _writeCoEData(AMSAddr, Index, SubIndex, ADR(Value), SIZEOF(Value));
END_METHOD

(*
Purpose
=======

This function is writing a real object via SDO.

*)
METHOD writeCoEDataREAL : EFieldbusQueryResult
VAR_INPUT CONSTANT
	AMSAddr				: AMSADDR;	
END_VAR
VAR_INPUT
	Index				: UINT;
	SubIndex			: BYTE;
	Value 				: REAL;
END_VAR

writeCoEDataREAL := _writeCoEData(AMSAddr, Index, SubIndex, ADR(Value), SIZEOF(Value));
END_METHOD

(*
Purpose
=======

This function is writing a sint object via SDO.

*)
METHOD writeCoEDataSINT : EFieldbusQueryResult
VAR_INPUT CONSTANT
	AMSAddr				: AMSADDR;	
END_VAR
VAR_INPUT
	Index				: UINT;
	SubIndex			: BYTE;
	Value 				: SINT;
END_VAR

writeCoEDataSINT := _writeCoEData(AMSAddr, Index, SubIndex, ADR(Value), SIZEOF(Value));
END_METHOD

(*
Purpose
=======

This function is writing a udint object via SDO.

*)
METHOD writeCoEDataUDINT : EFieldbusQueryResult
VAR_INPUT CONSTANT
	AMSAddr				: AMSADDR;	
END_VAR
VAR_INPUT
	Index				: UINT;
	SubIndex			: BYTE;
	Value 				: UDINT;
END_VAR

writeCoEDataUDINT := _writeCoEData(AMSAddr, Index, SubIndex, ADR(Value), SIZEOF(Value));
END_METHOD

(*
Purpose
=======

This function is writing a word object via SDO.

*)
METHOD writeCoEDataUINT : EFieldbusQueryResult
VAR_INPUT CONSTANT
	AMSAddr				: AMSADDR;	
END_VAR
VAR_INPUT
	Index				: UINT;
	SubIndex			: BYTE;
	Value 				: WORD;
END_VAR

writeCoEDataUINT := _writeCoEData(AMSAddr, Index, SubIndex, ADR(Value), SIZEOF(Value));
END_METHOD

(*
Purpose
=======

This function is writing a ulint object via SDO.

*)
METHOD writeCoEDataULINT : EFieldbusQueryResult
VAR_INPUT CONSTANT
	AMSAddr				: AMSADDR;	
END_VAR
VAR_INPUT
	Index				: UINT;
	SubIndex			: BYTE;
	Value 				: ULINT;
END_VAR

writeCoEDataULINT := _writeCoEData(AMSAddr, Index, SubIndex, ADR(Value), SIZEOF(Value));
END_METHOD

(*
Purpose
=======

This function is writing a usint object via SDO.

*)
METHOD writeCoEDataUSINT : EFieldbusQueryResult
VAR_INPUT CONSTANT
	AMSAddr				: AMSADDR;	
END_VAR
VAR_INPUT
	Index				: UINT;
	SubIndex			: BYTE;
	Value 				: USINT;
END_VAR

writeCoEDataUSINT := _writeCoEData(AMSAddr, Index, SubIndex, ADR(Value), SIZEOF(Value));
END_METHOD

(*
Purpose
=======

This function is writing a word object via SDO.

*)
METHOD writeCoEDataWORD : EFieldbusQueryResult
VAR_INPUT CONSTANT
	AMSAddr				: AMSADDR;	
END_VAR
VAR_INPUT
	Index				: UINT;
	SubIndex			: BYTE;
	Value 				: WORD;
END_VAR

writeCoEDataWORD := _writeCoEData(AMSAddr, Index, SubIndex, ADR(Value), SIZEOF(Value));
END_METHOD

METHOD writeCoEValueArray : EFieldbusQueryResult
VAR_INPUT CONSTANT
	AMSAddr			: AMSADDR;
	Objects			: POINTER TO EthercatCoEObjectArray;	
	Values 			: POINTER TO EthercatCoEValueArray; 	
END_VAR
VAR_INPUT
	Exec			: BOOL;
	Index			: REFERENCE TO DINT := 0;	
END_VAR
VAR_INST
	state			: EthWriteCoEArraySM;
	N 				: DINT;
	result			: EFieldbusQueryResult;
	trigger			: R_TRIG;
END_VAR
trigger(CLK:=Exec);

IF NOT Exec THEN
	state := 0;
END_IF

CASE state OF
	EthWriteCoEArraySM.IDLE: 	
		writeCoEValueArray := EFieldbusQueryResult.BUSY;
		IF trigger.Q THEN
			state := EthWriteCoEArraySM.INCR;
			N := -1;
		END_IF
		
	EthWriteCoEArraySM.WRITE: 
		writeCoEValueArray := EFieldbusQueryResult.BUSY;
		CASE Objects^[N].tclass OF
			EthTypes.TBYTE:
				result := writeCoEDataBYTE(AMSAddr, Objects^[N].idx, Objects^[N].sidx, Values^[N].VBYTE);
			EthTypes.TWORD:
				result := writeCoEDataWORD(AMSAddr, Objects^[N].idx, Objects^[N].sidx, Values^[N].VWORD);
			EthTypes.TDWORD:
				result := writeCoEDataDWORD(AMSAddr, Objects^[N].idx, Objects^[N].sidx, Values^[N].VDWORD);
			EthTypes.TLWORD:
				result := writeCoEDataLWORD(AMSAddr, Objects^[N].idx, Objects^[N].sidx, Values^[N].VLWORD);
			EthTypes.TSINT:
				result := writeCoEDataSINT(AMSAddr, Objects^[N].idx, Objects^[N].sidx, Values^[N].VSINT);
			EthTypes.TUSINT:
				result := writeCoEDataUSINT(AMSAddr, Objects^[N].idx, Objects^[N].sidx, Values^[N].VUSINT);
			EthTypes.TINT:
				result := writeCoEDataINT(AMSAddr, Objects^[N].idx, Objects^[N].sidx, Values^[N].VINT);
			EthTypes.TUINT:
				result := writeCoEDataUINT(AMSAddr, Objects^[N].idx, Objects^[N].sidx, Values^[N].VUINT);
			EthTypes.TDINT:
				result := writeCoEDataDINT(AMSAddr, Objects^[N].idx, Objects^[N].sidx, Values^[N].VDINT);
			EthTypes.TUDINT:
				result := writeCoEDataUDINT(AMSAddr, Objects^[N].idx, Objects^[N].sidx, Values^[N].VUDINT);
			EthTypes.TLINT:
				result := writeCoEDataLINT(AMSAddr, Objects^[N].idx, Objects^[N].sidx, Values^[N].VLINT);
			EthTypes.TULINT:
				result := writeCoEDataULINT(AMSAddr, Objects^[N].idx, Objects^[N].sidx, Values^[N].VULINT);
			EthTypes.TREAL:
				result := writeCoEDataREAL(AMSAddr, Objects^[N].idx, Objects^[N].sidx, Values^[N].VREAL);
			EthTypes.TLREAL:
				result := writeCoEDataLREAL(AMSAddr, Objects^[N].idx, Objects^[N].sidx, Values^[N].VLREAL);
		END_CASE

		IF __ISVALIDREF(Index) THEN
			Index := N;
		END_IF

		CASE result OF
			EFieldbusQueryResult.FAIL:
				state := EthWriteCoEArraySM.ERROR;
			EFieldbusQueryResult.OK:
				state := EthWriteCoEArraySM.INCR;				
		END_CASE
	
	EthWriteCoEArraySM.INCR:
		writeCoEValueArray := EFieldbusQueryResult.BUSY;
		N := N + 1;
		IF N > Parameters.SizeOfEthCoEValues-1 OR Objects^[N].para = 16#FFFF_FFFF THEN
			state := EthWriteCoEArraySM.READY;
		ELSE
			state := EthWriteCoEArraySM.WRITE;
		END_IF
		
	EthWriteCoEArraySM.READY:
		writeCoEValueArray := EFieldbusQueryResult.OK;
		IF NOT Exec THEN
			state := EthWriteCoEArraySM.IDLE;
		END_IF

	EthWriteCoEArraySM.ERROR:		
		writeCoEValueArray := EFieldbusQueryResult.FAIL;
		IF NOT Exec THEN
			state := EthWriteCoEArraySM.IDLE;
		END_IF		
		
END_CASE
END_METHOD

END_FUNCTION_BLOCK

// Fieldbus/EthercatCU2508Stat
(*
	This Class is collecting Ethercat Master Port Frame Lost data. Only ports that are linked via IO link to AMSADDR
	are processed. The class is robust in the case the reference is not linked.  
*)
FUNCTION_BLOCK EthercatCU2508Stat
VAR_INPUT
	IO_In : REFERENCE TO CU2508StatIO_In;
END_VAR
VAR
	{attribute 'hide'} 
	masters 	: ARRAY[0..7] OF EthercatMasterStat; 
	{attribute 'hide'} 
	amsnetid	: ARRAY[0..7] OF T_AMSNETID;
	{attribute 'hide'} 
	_lostframes : ARRAY[0..7] OF UDINT;
	{attribute 'hide'} 
	N			: UDINT;
	{attribute 'hide'} 
	started 	: BOOL;
END_VAR

IF (NOT STARTED) THEN
 	IF __ISVALIDREF(IO_In) THEN
		FOR N := 0 TO 7 DO
			amsnetid[N] := F_CreateAMSNetId(nIds:=IO_In.addr[N]);
		END_FOR
		started := TRUE;
	END_IF
END_IF

IF __ISVALIDREF(IO_In) THEN
	FOR N := 0 TO 7 DO
		IF IO_In.addr[N][0] <> 0 THEN
			masters[N](amsaddr:=amsnetid[N]);
		END_IF
	END_FOR
END_IF;

{attribute 'TcRpcEnable'}
METHOD getLostFrames : UDINT
VAR_INPUT
	port : DINT;
END_VAR
IF port = LIMIT(0,port,7) THEN
	getLostFrames := _lostframes[port];
ELSE
	getLostFrames := 666666;	
END_IF
END_METHOD

{attribute 'TcRpcEnable'}
METHOD setNull : BOOL
VAR_INPUT
	port : UDINT;
END_VAR
IF port = LIMIT(0,port,7) THEN
	masters[port].setNull();
END_IF
END_METHOD

END_FUNCTION_BLOCK

// Fieldbus/EthercatMasterStat
{attribute 'hide_all_locals'}
FUNCTION_BLOCK EthercatMasterStat
VAR_INPUT
	amsaddr 	: REFERENCE TO T_AMSNETID;
END_VAR
VAR
	stat 		: FB_EcMasterFrameStatistic;
	clear		: FB_EcMasterFrameStatisticClearFrames;
	_lostFrames : UDINT; 
	_clearError	: BOOL;
	exec 		: BOOL;
	busy 		: BOOL;
	state		: DINT;
	timer		: TON;
END_VAR


IF _clearError THEN
	clear(
		sNetId 		:= amsaddr,
		bExecute 	:= TRUE,
		tTimeout	:= T#500MS,
		bBusy		=> busy
	);
ELSE
	stat(
		sNetId 			:= amsaddr,
		bExecute 		:= TRUE,
		tTimeout 		:= T#500MS,
		bBusy			=> busy
	);	
END_IF


timer(IN := state = 10, PT:= T#2S);

CASE state OF
	0: 
		state := 10;
		exec := FALSE;
		
	10:
		exec := TRUE;
		IF timer.Q AND (NOT busy) THEN
			IF NOT _clearError THEN
				_lostFrames := stat.nLostFrames;
			ELSE
				_clearError := FALSE;
			END_IF
			state := 20;
		END_IF
		
	20:
		exec := FALSE;
		state := 10;
END_CASE

{attribute 'monitoring':='call'}
{attribute 'TcRpcEnable'}
PROPERTY LostFrames : UDINT
GET
LostFrames := _lostFrames;
END_GET
END_PROPERTY

{attribute 'TcRpcEnable'}
METHOD setNull : BOOL
_clearError := True;
END_METHOD

END_FUNCTION_BLOCK

// IOHandler/IIOHandler
INTERFACE IIOHandler

METHOD ABSTRACT get : BOOL
VAR_INPUT
	io_in		: REFERENCE TO PVOID;
	io_out		: REFERENCE TO PVOID;
END_VAR
END_METHOD

END_INTERFACE

// IOHandler/IOHandler
(*
This abstract class makes it feasable to put IO on a global level
*)
{attribute 'hide_all_locals'}
FUNCTION_BLOCK ABSTRACT IOHandler Implements IIOHandler
VAR
	unittesting		: BOOL;
END_VAR

METHOD  FB_init : BOOL
VAR_INPUT
	bInitRetains	: BOOL; // if TRUE, the retain variables are initialized (warm start / cold start)
	bInCopyCode 	: BOOL;  // if TRUE, the instance afterwards gets moved into the copy code (online change)
	UnitTesting 	: BOOL;
END_VAR
THIS^.unittesting := UnitTesting;
END_METHOD

METHOD ABSTRACT get : BOOL
VAR_INPUT
	io_in		: REFERENCE TO PVOID;
	io_out		: REFERENCE TO PVOID;
END_VAR
(*

IF THIS^.unitTest THEN
	io_in := ADR(THIS^.ioout_test);
	io_out := ADR(THIS^.ioin_test);
ELSE
	io_in := ADR(THIS^.ioout);
	io_out := ADR(THIS^.ioin);
END_IF

*)
END_METHOD

END_FUNCTION_BLOCK

// Math/CosineRuleKnownAllSides
(*
Purpose
=======
This function calculates the angle A given all sides of a triangle
Returns value in Radians

Usage
======
Check side placements, wrong placements result in output for angle B or C
Sketchup on dimensional sketch and save example used of reference.
NOTE: make sure that all input is of same unit size.
b & c can't be 0
a + b must be > c

Methods And Properties
======================
*)
FUNCTION CosineRuleKnownAllSides : LREAL
{attribute 'hide_all_locals'}
VAR_INPUT
	a : LREAL;	//	Left side of angle
	b : LREAL;	//	Rigth side of angle 
	c : LREAL;	//	Opposite side of the angle we want
END_VAR

VAR
	angle : LREAL;
    a2b2: LREAL; // Value of a^2 + b^2
    c2: LREAL; // Value of c^2
    denominator: LREAL; // Denominator of the formula
END_VAR

IF b * a <> 0 THEN // no DBZ check
	// Calculate a^2 + b^2
    a2b2 := a*a + b*b;
    
    // Calculate c^2
    c2 := c*c;
    
    // Calculate the denominator of the formula
    denominator := 2*a*b;
    
    // Calculate angle using the formula. NOTE: Return angle in radians
    angle := ACOS((a2b2 - c2) / denominator);
ELSE
	angle:= 0;
END_IF
CosineRuleKnownAllSides := angle;

END_FUNCTION

// Math/CosineRuleKnownAnAngle
(*
Purpose
=======
This function calculates the side c given angle C and the rest of triangle sides

Usage
======
Check side or angle placements, 
wrong placements result in output for wrong side or not a value to the triangle at all
Sketchup on dimensional sketch and save example used of reference.

Methods And Properties
======================
*)
{attribute 'hide_all_locals'}
FUNCTION CosineRuleKnownAnAngle : LREAL
VAR_INPUT
	a : LREAL;	//	Side
	b : LREAL;	//	Side
	c : LREAL;	//	opposite side of angle c
END_VAR

CosineRuleKnownAnAngle := SQRT(EXPT(a,2) + EXPT(b,2) - (2*a*b*COS(c)));

END_FUNCTION

// Math/HorizontalLength
(*
Purpose
=======
This function calculates the Length of a body part in handling equipment
when building handling equipment with multiple body parts it's nice to separate, 
them before adding them together. This makes developing and troubleshooting easier.

Methods And Properties
======================
*)
{attribute 'hide_all_locals'}
FUNCTION HorizontalLength : LREAL
VAR_INPUT
	angle : LREAL;	//	leg angle reference to horizontal line [rad]
	length : LREAL;	//	length of the leg
END_VAR

HorizontalLength := (COS(angle) * length) * (-1);

END_FUNCTION

// Math/Signum
(*
Purpose
=======
This function calculates the signum of a numeric value

Methods And Properties
======================
*)
{attribute 'hide_all_locals'}
FUNCTION Signum : LREAL
VAR_INPUT
	x : LREAL;
END_VAR

Signum := SEL(x>=0.0, -1.0, 1.0);

END_FUNCTION

// Math/VerticalHeight
(*
Purpose
=======
This function calculates the Height of a body part in handling equipment
when building handling equipment with multiple body parts it's nice to separate, 
them before adding them together. This makes developing and troubleshooting easier.

Methods And Properties
======================
*)
{attribute 'hide_all_locals'}
FUNCTION VerticalHeight : LREAL
VAR_INPUT
	angle : LREAL;	//	leg angle reference to horizontal line [rad]
	length : LREAL;	//	length of the leg
END_VAR

VerticalHeight := SIN(angle) * length;

END_FUNCTION

// MRU/IMRUReader
(*
Purpose
=======
This is the interface definition providing an interface for the MRU class to read MRU values


Methods And Properties
======================
*)
INTERFACE IMRUReader

{attribute 'TcRpcEnable'}
PROPERTY DataAvailable : BOOL
GET
END_GET
END_PROPERTY

{attribute 'TcRpcEnable'}
METHOD getData : BOOL
VAR_INPUT
	NMEAdata : REFERENCE TO TNMEAsentence;
END_VAR
END_METHOD

END_INTERFACE

// MRU/MRU
(*
Purpose
=======
This is a MRU class.  The class is reading a NMEA sentence from an object providing 
an IMRUReader interface and decodes the NMEA date by the NMEAParser class. The data 
is then transformed to the position of interest by a transformation function. Up to 
ten points can be defined  

Features
========

#. Automatic transformation of NMEA data to point of interests

Methods And Properties
======================
*)
{attribute 'no_explicit_call' := 'do not call this POU directly'} 
{attribute 'hide_all_locals'}
FUNCTION_BLOCK MRU
VAR
	Config : ConfigMRU;
	parser : NMEAParser;
	acceleration, velocity, position : LREAL; // MRU values
	pitch, roll, pitch_rate, roll_rate : LREAL; // MRU values
	_acceleration, _position, _velocity : LREAL; // transformed values
END_VAR

{attribute 'TcRpcEnable'}
METHOD getValues : BOOL
VAR_INPUT
	Position 		: REFERENCE TO LREAL;
	Velocity 		: REFERENCE TO LREAL;
	Acceleration 	: REFERENCE TO LREAL;
END_VAR
Position := THIS^._position;
Velocity := THIS^._velocity;
Acceleration := THIS^._acceleration;
END_METHOD

// Attention input for angles are now in radian!!! 
//
// Functional description:
//
//This function is used to calculate the crane tip movement from the MRU heave, 
//velocity, pitch and roll values. The MRU is setup to provide the values for the 
//top center of the crane king (measuring point). Crane tip XYZ coordinates are 
//relative to this point.
//

//The function takes the MRU heave and velocity values and adds corrections for 
//pitch and roll motion around the MRU measuring point. The calculation of the
//velocity and acceleration is adjustable (delta t for differentiation) and can be
//filtered (using 1st order filter). 
//
//Coordinate inputs are filtered (ramped) to avoid sudden jumps in heave and 
//velocity outputs.
//
//Input definitions:
//
//ifX                   X vector positive horisontal pointing forward (m)
//ifY                   Y vector is positive horisontal pointing port (m)
//ifZ                   Z vektor is positive vertical pointing up (m)
//ifMRU_Heave           Heave positive down (m)
//ifMRU_Velocity        Velocity positive down (m/s)
//ifMRU_Pitch           Pitch angle positive if lifting the bow (rad)
//ifMRU_Roll            Roll angle positive if leaning to stb side (rad)
//ifDeltaT_XXX          Delta T is the minimum delta time used in differentiation
//ifAlpha_XXX           Alpha is a filtering constant (1 means no filter)
//ifMRU_Pitch_Rate      Digital MRU pitch angle speed (positive lifting bow)(rad/s)
//ifMRU_Roll_Rate       Digital MRU roll angle speed (positive leaning stb) (rad/s)
//
//Output definitions:
//
//
//qfTrue_Heave          True heave positive down (m)
//qfTrue_Velocity       True velocity positive down (m/s)
//qfTrue_Accel          True acceleration positive down (m/s^2)   
//qfTrue_Velocity_MRU   True velocity positive down based on digital MRU  (m/s)
METHOD transform : BOOL
VAR_INPUT
    ifX                     :LREAL:= 0.0;    //POI vector X (X-axis forward) (m)
    ifY                     :LREAL:= 0.0;    //POI vector Y (Y-axis port) (m)
    ifZ                     :LREAL:= 0.0;    //POI vector Z (Z-axis up) (m)
    ifMRU_Heave             :LREAL:= 0.0;    //MRU heave position (positive down) (m)
    ifMRU_Velocity          :LREAL:= 0.0;    //MRU heave velocity (positive down) (m/s)
    ifMRU_Pitch             :LREAL:= 0.0;    //MRU pitch angle (positive lifting bow)(rad)
    ifMRU_Roll              :LREAL:= 0.0;    //MRU roll angle (positive leaning stb) (rad)
    ifMRU_Pitch_Rate        :LREAL:= 0.0;    //MRU pitch angle speed (positive lifting bow)(rad/s)(
    ifMRU_Roll_Rate         :LREAL:= 0.0;    //MRU roll angle speed (positive leaning stb) (rad/s)
    ifDeltaT_Vel            :LREAL:= 0.0;    //True velocity calculation delta time (s)
    ifAlpha_Vel             :LREAL:= 0.0;    //True velocity filter constant (0 to 1, 1 = no filter)
    ifDeltaT_Acc            :LREAL:= 0.0;    //True acceleration calculation delta time (s)
    ifAlpha_Acc             :LREAL:= 0.0;    //True acceleration filter constant (0 to 1, 1 = no filter)
    ifCycleTime             :LREAL:= 0.0;    //Block call cycle time (s)   	
END_VAR

VAR_OUTPUT  //Block outputs
    qfTrue_Heave            :LREAL;          //Calculated output value (true heave position) (m)
    qfTrue_Velocity         :LREAL;          //Calculated output value (true heave velocity) (m/s)
    qfTrue_Accel            :LREAL;          //Calculated output value (true heave acceleration) (m/s^2)
    qfTrue_Velocity_MRU     :LREAL;          //Calculated output value based on MRU (true heave velocity) (m/s)  
END_VAR
VAR_INST //Static variables
    fLastTrueHeave          :LREAL;
    fLastMRUHeave           :LREAL;
    fLastX                  :LREAL;
    fLastY                  :LREAL;
    fLastZ                  :LREAL;
    fLastDeltaVelocity      :LREAL;
    fVelocityTimer          :LREAL;
    fDeltaVelocity          :LREAL;
    fAccelTimer             :LREAL;
    fAcceleration           :LREAL;
    fLastVelocity           :LREAL;
    fLastAcceleration       :LREAL;
END_VAR
VAR  
    fRollCorr               :LREAL;          //Roll correction in x direction
    fPitchCorr              :LREAL;          //Pitch correction in x direction
    fRoll                   :LREAL;          //Roll in Radians
    fPitch                  :LREAL;          //Pitch in Radians
    fCurrX                  :LREAL;
    fCurrY                  :LREAL;
    fCurrZ                  :LREAL;
    tfMRU_Roll_Rate_rad     :LREAL;
    tfMRU_Pitch_Rate_rad    :LREAL;
    fRollCorr_MRU           :LREAL;          //Roll correction in x direction based on MRU
    fPitchCorr_MRU          :LREAL;          //Pitch correction in x direction based on MRU
    tfTrue_Velocity         :LREAL;
    D_W                     :DWORD;
END_VAR
VAR CONSTANT  
    Pi 						: LREAL := p7type.math.PI;
END_VAR

// Input mapping

fCurrX:= ifX;
fCurrY:= ifY;
fCurrZ:= ifZ;

// Input coordinate filtering. These coordinates 
IF ifCycleTime > 0.0 THEN
	IF (fCurrX - fLastX) / ifCycleTime > 0.5 THEN
		fCurrX:= fLastX + 0.5 * ifCycleTime;
	ELSIF (fCurrX - fLastX) / ifCycleTime < -0.5 THEN
		fCurrX:= fLastX - 0.5 * ifCycleTime;
	END_IF;
	IF (fCurrY - fLastY) / ifCycleTime > 0.5 THEN
		fCurrY:= fLastY + 0.5 * ifCycleTime;
	ELSIF (fCurrY - fLastY) / ifCycleTime < -0.5 THEN
		fCurrY:= fLastY - 0.5 * ifCycleTime;
	END_IF;
	IF (fCurrZ - fLastZ) / ifCycleTime > 0.5 THEN
		fCurrZ:= fLastZ + 0.5 * ifCycleTime;
	ELSIF (fCurrZ - fLastZ) / ifCycleTime < -0.5 THEN
		fCurrZ:= fLastZ - 0.5 * ifCycleTime;
	END_IF;
END_IF;

// Don't Convert degrees to radians since MRU from Kongsberg is delivering Radian
fPitch:= ifMRU_Pitch;
fRoll:= ifMRU_Roll;
tfMRU_Pitch_Rate_rad := ifMRU_Pitch_Rate;
tfMRU_Roll_Rate_rad := ifMRU_Roll_Rate;

// Calculate pitch correction value
IF fCurrX = 0.0 THEN
	fPitchCorr:= fCurrZ * (1.0 - SIN((Pi/2) + fPitch));
ELSIF fCurrX > 0.0 THEN
	fPitchCorr:= fCurrZ - SQRT(EXPT(fCurrX,2) + EXPT(fCurrZ,2)) * SIN(ATAN(fCurrZ/fCurrX) + fPitch);
ELSE
	fPitchCorr:= fCurrZ + SQRT(EXPT(fCurrX,2) + EXPT(fCurrZ,2)) * SIN(ATAN(fCurrZ/fCurrX) + fPitch);
END_IF;

    
// Calculate roll correction value
IF fCurrY = 0.0 THEN
	fRollCorr:= fCurrZ * (1.0 - SIN((Pi/2) + fRoll));
ELSIF fCurrY > 0.0 THEN
	fRollCorr:= fCurrZ - SQRT(EXPT(fCurrY,2) + EXPT(fCurrZ,2)) * SIN(ATAN(fCurrZ/fCurrY) + fRoll);
ELSE
	fRollCorr:= fCurrZ + SQRT(EXPT(fCurrY,2) + EXPT(fCurrZ,2)) * SIN(ATAN(fCurrZ/fCurrY) + fRoll);
END_IF;


// Calculate crane tip heave position
qfTrue_Heave:= ifMRU_Heave + fPitchCorr + fRollCorr;

// Calculate delta velocity
fVelocityTimer:= fVelocityTimer + ifCycleTime;

IF fVelocityTimer >= ifDeltaT_Vel AND fVelocityTimer > 0.0 THEN   
	fDeltaVelocity:= ((qfTrue_Heave - ifMRU_Heave) - (fLastTrueHeave - fLastMRUHeave)) / fVelocityTimer;
	fVelocityTimer:= 0.0;
	fLastTrueHeave:= qfTrue_Heave;
	fLastMRUHeave:= ifMRU_Heave;
END_IF;

// Filter delta velocity
fDeltaVelocity:= ifAlpha_Vel*fDeltaVelocity + (1-ifAlpha_Vel)*fLastDeltaVelocity;

// True velocity
tfTrue_Velocity:= ifMRU_Velocity + fDeltaVelocity;


// Check for invalid number and store current values for next scan
D_W := LREAL_TO_DWORD(tfTrue_Velocity) AND DWORD#16#7F800000;
IF NOT (D_W = DWORD#16#7F800000) THEN
	fLastDeltaVelocity:= fDeltaVelocity;
	qfTrue_Velocity:= tfTrue_Velocity;
ELSE
	fLastDeltaVelocity:= 0.0;
	qfTrue_Velocity := 0.0;
END_IF;



// Calculate acceleration
fAccelTimer:= fAccelTimer + ifCycleTime;
IF fAccelTimer >= ifDeltaT_Acc AND fAccelTimer > 0.0 THEN
	fAcceleration:= (ifMRU_Velocity - fLastVelocity) / fAccelTimer;
	fAccelTimer:= 0.0;
	fLastVelocity:= ifMRU_Velocity;
END_IF;

// Filter acceleration
qfTrue_Accel:= ifAlpha_Acc*fAcceleration + (1-ifAlpha_Acc)*fLastAcceleration;

// Store current values for next scan
fLastDeltaVelocity:= fDeltaVelocity;
fLastAcceleration:= qfTrue_Accel;
fLastX:= fCurrX;
fLastY:= fCurrY;
fLastZ:= fCurrZ;

// Calculate pitch correction value
IF fCurrX = 0.0 THEN
	fPitchCorr_MRU:= fCurrZ * (1.0 - SIN((Pi/2) + fPitch));
ELSIF fCurrX > 0.0 THEN
	fPitchCorr_MRU:= fCurrZ - SQRT(EXPT(fCurrX,2) + EXPT(fCurrZ,2)) * SIN(ATAN(fCurrZ/fCurrX) + tfMRU_Pitch_Rate_rad);
ELSE
	fPitchCorr_MRU:= fCurrZ + SQRT(EXPT(fCurrX,2) + EXPT(fCurrZ,2)) * SIN(ATAN(fCurrZ/fCurrX) + tfMRU_Pitch_Rate_rad);
END_IF;


// Calculate roll correction value
IF fCurrY = 0.0 THEN
	fRollCorr_MRU:= fCurrZ * (1.0 - SIN((Pi/2) + fRoll));
ELSIF fCurrY > 0.0 THEN
	fRollCorr_MRU:= fCurrZ - SQRT(EXPT(fCurrY,2) + EXPT(fCurrZ,2)) * SIN(ATAN(fCurrZ/fCurrY) + tfMRU_Roll_Rate_rad);
ELSE
	fRollCorr_MRU:= fCurrZ + SQRT(EXPT(fCurrY,2) + EXPT(fCurrZ,2)) * SIN(ATAN(fCurrZ/fCurrY) + tfMRU_Roll_Rate_rad);
END_IF;

qfTrue_Velocity_MRU := ifMRU_Velocity + fPitchCorr_MRU + fRollCorr_MRU;
END_METHOD

(*
Purpose
=======
This method is updating MRU data and must be called cyclically. Best practice would be call
update() twice as fast as the MRU cycle time

*)
METHOD update : BOOL
VAR_INPUT
	Config : REFERENCE TO ConfigMRU;
	datareader : IMRUreader;
END_VAR
VAR_INST
	sentence 	: TNMEAsentence;
	started 	: BOOL; 
END_VAR
IF NOT started THEN
	started := TRUE; 
	parser.setFieldsOfInterest('RRRRRRR'); (* Velocity, Position, Acceleration, Pitch,
											Pitch Rate, Roll, Roll Rate *)
END_IF

THIS^.Config := Config;

update := FALSE;
IF datareader.DataAvailable THEN
	datareader.getData(NMEAdata := sentence);
	IF parser.parse(sentence) THEN
		velocity := SEL(Config.Option_Reverse_Velocity, parser.getRealField(0), -parser.getRealField(0));
		position := SEL(Config.Option_Reverse_Position, parser.getRealField(1), -parser.getRealField(1));
		acceleration := SEL(Config.Option_Reverse_Acceleration, parser.getRealField(2), -parser.getRealField(2));
		pitch  := SEL(Config.Option_Reverse_Ritch, parser.getRealField(3), -parser.getRealField(3));
		pitch_rate  := SEL( Config.Option_Reverse_Ritch, parser.getRealField(4), -parser.getRealField(4));
		roll := SEL(Config.Option_Reverse_Roll, parser.getRealField(5), -parser.getRealField(5));
		roll_rate  := SEL(Config.Option_Reverse_Roll, parser.getRealField(6), -parser.getRealField(6));
		
		IF Config.Option_MRUSet >= 0 THEN 
			transform(
				ifX :=  Config.PosX[Config.Option_MRUSet],
				ifY :=  Config.PosY[Config.Option_MRUSet],
				ifZ :=  Config.PosZ[Config.Option_MRUSet],
				ifMRU_Heave := THIS^.position,
				ifMRU_Velocity := THIS^.velocity,
				ifMRU_Pitch := THIS^.pitch,
				ifMRU_Roll := THIS^.roll,
				ifMRU_Roll_Rate := THIS^.roll_rate,
				ifMRU_Pitch_Rate := THIS^.pitch_rate,
				ifDeltaT_Vel := Config.CycleTime,
				ifAlpha_Vel := 1.0,
				ifDeltaT_Acc := Config.CycleTime,
				ifAlpha_Acc := 1.0,
				ifCycleTime := Config.CycleTime,
				qfTrue_Heave => _Position,
				qfTrue_Velocity => _Velocity,
				qfTrue_Accel => _Acceleration
			);
		ELSE
			Position := THIS^.position; 
			Velocity := THIS^.velocity; 
			Acceleration := THIS^.acceleration; 
		END_IF;		
		update := TRUE;
	ELSE
	 	update := FALSE; 
	END_IF
END_IF
END_METHOD

END_FUNCTION_BLOCK

// NMEA/NMEAParser
{attribute 'no_explicit_call' := 'do not call this POU directly'}
(*
Purpose
=======
This class parses an NMEA0183 sentence with up to 32 field excluding the header. 
The parse method returns a bool value to indicate success. Up to 32 fields will 
be returned. 

How To
======
First setup the fields of interests and run the parse method. The field indices 
are equal to the field position.  

Attention: Any $ char has to be escaped with a $ in the case a constant is
used. 

Example 
=======
nmea.setFieldsOfInterests('IIIRS');
nmea.parse('$$PRAP,22,33,4,3.1,Hello*65');
header := nmea.getHeader(); // PRAP
result1 := nmea.getIntField(0); // 22
result2 := nmea.getIntField(1); // 33
result3 := nmea.getIntField(2); // 4
result4 := nmea.getRealField(3); // 3.1
result5 := nmea.getStringField(5); // Hello

Methods And Properties
======================
*)
{attribute 'hide_all_locals'}
FUNCTION_BLOCK NMEAParser
VAR
	header 				: STRING(5);
	sentenceStructure 	: TNMEAStructDescription;
	stringFields 		: ARRAY[0..31] OF TNMEAstring;
	intFields			: ARRAY[0..31] OF TNMEAint;
	realFields			: ARRAY[0..31] OF TNMEAreal;
END_VAR
VAR CONSTANT
	TNMEAstringsz 		: INT := 64;
END_VAR

METHOD PRIVATE _hexChkSum_to_byte : BYTE
VAR_INPUT
	data : STRING(2);
END_VAR
VAR
	sum, a ,b : BYTE;
	pbyte : POINTER TO BYTE;
END_VAR

pbyte := ADR(data);

a := pbyte^ - 48; 
pbyte := pbyte + 1;
b := pbyte^ - 48; 

IF a > 9 THEN
	a := a - 7; 
END_IF

IF b > 9 THEN
	b := b - 7;
END_IF

_hexChkSum_to_byte := a * BYTE#16 + b;
END_METHOD

METHOD PRIVATE _incp : POINTER TO BYTE
VAR_IN_OUT
	p : POINTER TO BYTE;
END_VAR
p := p + 1;
END_METHOD

METHOD calcChkSum : BOOL
VAR_IN_OUT CONSTANT
	Sentence : TNMEAsentence;	
END_VAR
VAR_IN_OUT
	Checksum : BYTE;
END_VAR
VAR
	msglen : INT;
	N : INT;
	chksum : BYTE;
	char : BYTE; 
	pbyte : POINTER TO BYTE;
	x : BYTE;
END_VAR
Checksum := 0;
msglen := LEN(Sentence);


pbyte := ADR(Sentence)+1;

FOR N := 2 TO msglen DO
	IF (pbyte^=42) THEN // Char *
		EXIT;
	ELSIF  (pbyte^=10) OR (pbyte^=13) THEN // Chars NL and CR
		calcChkSum := FALSE;
		RETURN;
	END_IF
	
	Checksum := Checksum XOR pbyte^;
	pbyte := pbyte + 1;
END_FOR

calcChkSum := TRUE;
END_METHOD

METHOD getChkSumFromSentence : BOOL
VAR_IN_OUT CONSTANT
	Sentence : TNMEAsentence;
END_VAR
VAR_IN_OUT
	Checksum : USINT;	
END_VAR
VAR_INST
	msglen : INT;
	char : BYTE;
	N : INT; 
	pbyte : POINTER TO BYTE;
	ps : POINTER TO STRING;
	c1, c2 : BYTE;
	chksumascii : STRING(2) := '00';
END_VAR
Checksum := 0;
msglen := LEN(Sentence);
pbyte := ADR(Sentence) + INT_TO_DWORD(msglen) - 1;

IF msglen < 11 THEN 
	getChkSumFromSentence := FALSE;
	RETURN;
END_IF

getChkSumFromSentence := FALSE;
FOR N := msglen TO 4 BY -1 DO
	IF pbyte^ = 42 THEN // Char * 
		pbyte := pbyte + 1;
		getChkSumFromSentence := TRUE;
		EXIT;
	ELSIF N = 4 THEN
		getChkSumFromSentence := FALSE;
		RETURN;		
	END_IF

	pbyte := pbyte - 1;	
END_FOR

ps := pbyte;
chksumascii := LEFT(ps^, 2);
Checksum := _hexChkSum_to_byte(chksumascii);

getChkSumFromSentence := TRUE;
END_METHOD

METHOD getHeader : STRING(5)
getHeader := THIS^.header;
END_METHOD

METHOD getIntField : TNMEAint
VAR_INPUT
	FieldNo : UINT;
END_VAR
getIntField := THIS^.intFields[FieldNo];
END_METHOD

METHOD getRealField : TNMEAreal
VAR_INPUT
	FieldNo : UINT;
END_VAR
getRealField := THIS^.realFields[FieldNo];
END_METHOD

METHOD getStringField : TNMEAstring
VAR_INPUT
	FieldNo : UINT;
END_VAR
getStringField := THIS^.stringFields[FieldNo];
END_METHOD

(*
Purpose
=======
Parse a NMEA0183 sentence and return TRUE in the case of a success. Buffer overflow 
was prevented by sizing strings to the worst case and checking the length. 

